__TRY
	_Ancestor.AddChildActivity(activity := _Ancestor);
__CATCH(exceptionCode)
	exception := TOF_Core.ExceptionManager.GetLastException(
		exceptionCode := exceptionCode,
		catchPointNamespaceName := NamespaceName,
		catchPointPOUName := __POUNAME(),
		catchPointPosition := __POSITION()
	);
	caught := __QUERYINTERFACE(exception, attachmentException);
__ENDTRY

assertions.ThatBool(actual := caught, message := "Self attachment must be rejected").IsTrue();
_Ancestor.AddChildActivity(activity := _Descendant);
caught := FALSE;

__TRY
	_Descendant.AddChildActivity(activity := _Ancestor);
__CATCH(exceptionCode)
	exception := TOF_Core.ExceptionManager.GetLastException(
		exceptionCode := exceptionCode,
		catchPointNamespaceName := NamespaceName,
		catchPointPOUName := __POUNAME(),
		catchPointPosition := __POSITION()
	);
	caught := __QUERYINTERFACE(exception, attachmentException);
__ENDTRY

assertions.ThatBool(actual := caught, message := "Ancestor attachment must be rejected").IsTrue();

_Pick.AddBranch(condition := _PickFirstCondition, activity := _PickFirstActivity);
caught := FALSE;

__TRY
	_Pick.AddBranch(condition := _PickFirstCondition, activity := _PickSecondActivity);
__CATCH(exceptionCode)
	exception := TOF_Core.ExceptionManager.GetLastException(
		exceptionCode := exceptionCode,
		catchPointNamespaceName := NamespaceName,
		catchPointPOUName := __POUNAME(),
		catchPointPosition := __POSITION()
	);
	caught := __QUERYINTERFACE(exception, attachmentException);
__ENDTRY

assertions.ThatBool(actual := caught, message := "A condition cannot occupy two branch slots").IsTrue();
caught := FALSE;

__TRY
	_Pick.AddBranch(condition := _PickSecondCondition, activity := _PickFirstActivity);
__CATCH(exceptionCode)
	exception := TOF_Core.ExceptionManager.GetLastException(
		exceptionCode := exceptionCode,
		catchPointNamespaceName := NamespaceName,
		catchPointPOUName := __POUNAME(),
		catchPointPosition := __POSITION()
	);
	caught := __QUERYINTERFACE(exception, attachmentException);
__ENDTRY

assertions.ThatBool(actual := caught, message := "An activity cannot occupy two branch slots").IsTrue();
actualElement := _PickSecondCondition.Parent;
assertions.ThatBool(
	actual := actualElement = 0,
	message := "Rejected pairs must not attach the unused condition"
).IsTrue();
actualElement := _PickSecondActivity.Parent;
assertions.ThatBool(
	actual := actualElement = 0,
	message := "Rejected pairs must not attach the unused activity"
).IsTrue();
_Pick.AddBranch(condition := _PickSecondCondition, activity := _PickSecondActivity);
_PickFirstActivity.completeRunning := TRUE;
_Pick.RequestStart();
assertions.ThatDInt(
	actual := _Pick.CurrentBranchIndex,
	message := "The original first pair must retain priority"
).ToBe(expected := 0);
assertions.ThatDInt(
	actual := _PickFirstActivity.startCount,
	message := "The first branch activity must start"
).ToBe(expected := 1);
assertions.ThatDInt(
	actual := _PickSecondActivity.startCount,
	message := "The second branch must remain unstarted"
).ToBe(expected := 0);

_SequenceFirst.completeRunning := TRUE;
_SequenceSecond.completeRunning := TRUE;
_Sequence.RequestStart();
_Sequence.Execute();
assertions.ThatBool(
	actual := _Sequence.State = TOF_Workflow.WORKFLOW_ELEMENT_STATE.PASSIVE_COMPLETED,
	message := "The original two valid slots must complete"
).IsTrue();
assertions.ThatDInt(
	actual := _SequenceFirst.startCount,
	message := "First child must start once"
).ToBe(expected := 1);
assertions.ThatDInt(
	actual := _SequenceSecond.startCount,
	message := "Second child must start once"
).ToBe(expected := 1);

_Sequence.RequestReset();
_Pick.RequestReset();
assertions.ThatBool(
	actual := _Sequence.CurrentActivityIndex = TOF_Workflow.Workflows.NO_SELECTED_ACTIVITY_INDEX,
	message := "Reset sequence must expose the documented absent-selection sentinel"
).IsTrue();
assertions.ThatBool(
	actual := _Pick.CurrentBranchIndex = TOF_Workflow.Workflows.NO_SELECTED_ACTIVITY_INDEX,
	message := "Reset branch selection must expose the same absent-selection sentinel"
).IsTrue();
END_METHOD

(*!
<summary>Preserves task internal-abort diagnostics while stopping.</summary>
<description>
Uses independently prepared persistent fixtures. Expected failures are checked by exception interface;
ordinary unexpected exceptions leave fixture ownership with the suite.
</description>
<param name="assertions">Valid assertion context borrowed from the active case.</param>
*)
METHOD PRIVATE testTaskAbortDuringSuspend
VAR_INPUT
	assertions : REFERENCE TO TOF_Testing.Assertions;
END_VAR
_SuspendAbortActivity.Configure(task := _SuspendAbortTask);
_SuspendAbortWorkflow.SetRootActivity(rootActivity := _SuspendAbortActivity);
_SuspendAbortWorkflow.RequestStart();
_SuspendAbortTask.processingResult := TOF_Tasks.TASK_PROCESSING_STATE.ABORTED;
_SuspendAbortWorkflow.RequestSuspend();
assertions.ThatBool(
	actual := _SuspendAbortActivity.State = TOF_Workflow.WORKFLOW_ELEMENT_STATE.PASSIVE_HALTED,
	message := "An internal abort while suspending must remain HALTED"
).IsTrue();
assertions.ThatWideString(
	actual := _SuspendAbortActivity.HaltReason,
	message := "The task abort reason must survive adapter translation"
).ToBe(expected := "Controlled task internal abort");
_SuspendAbortWorkflow.RequestReset();
END_METHOD

(*!
<summary>Preserves successful task completion when work finishes during suspension.</summary>
<description>
Uses independently prepared persistent fixtures. Expected failures are checked by exception interface;
ordinary unexpected exceptions leave fixture ownership with the suite.
</description>
<param name="assertions">Valid assertion context borrowed from the active case.</param>
*)
METHOD PRIVATE testTaskCompletionDuringSuspend
VAR_INPUT
	assertions : REFERENCE TO TOF_Testing.Assertions;
END_VAR
_SuspendDoneActivity.Configure(task := _SuspendDoneTask);
_SuspendDoneWorkflow.SetRootActivity(rootActivity := _SuspendDoneActivity);
_SuspendDoneWorkflow.RequestStart();
_SuspendDoneTask.processingResult := TOF_Tasks.TASK_PROCESSING_STATE.DONE;
_SuspendDoneWorkflow.RequestSuspend();
assertions.ThatBool(
	actual := _SuspendDoneActivity.State = TOF_Workflow.WORKFLOW_ELEMENT_STATE.PASSIVE_COMPLETED,
	message := "Work completed during suspension must retain its completion outcome"
).IsTrue();
_SuspendDoneWorkflow.RequestReset();
END_METHOD

(*!
<summary>Reports a task processing failure during suspension as an activity failure.</summary>
<description>
Uses independently prepared persistent fixtures. Expected failures are checked by exception interface;
ordinary unexpected exceptions leave fixture ownership with the suite.
</description>
<param name="assertions">Valid assertion context borrowed from the active case.</param>
*)
METHOD PRIVATE testTaskFailureDuringSuspend
VAR_INPUT
	assertions : REFERENCE TO TOF_Testing.Assertions;
END_VAR
_SuspendFailureActivity.Configure(task := _SuspendFailureTask);
_SuspendFailureWorkflow.SetRootActivity(rootActivity := _SuspendFailureActivity);
_SuspendFailureWorkflow.RequestStart();
_SuspendFailureTask.processingResult := TOF_Tasks.TASK_PROCESSING_STATE.ERROR;
_SuspendFailureWorkflow.RequestSuspend();

assertions.ThatBool(
	actual := _SuspendFailureTask.State.Stopped,
	message := "The failed task must reach STOPPED"
).IsTrue();
assertions.ThatBool(
	actual := _SuspendFailureActivity.State = TOF_Workflow.WORKFLOW_ELEMENT_STATE.PASSIVE_FAILED,
	message := "Task failure while suspending must not be reported as SUSPENDED"
).IsTrue();
assertions.ThatBool(
	actual := _SuspendFailureWorkflow.FailError.HasError,
	message := "Failure diagnostics must be retained"
).IsTrue();
_SuspendFailureWorkflow.RequestReset();
END_METHOD

(*!
<summary>
Keeps servicing cancellation through release and exposes a release failure with explicit resource recovery.
</summary>
<description>
Uses independently prepared persistent fixtures. Expected failures are checked by exception interface;
ordinary unexpected exceptions leave fixture ownership with the suite.
</description>
<param name="assertions">Valid assertion context borrowed from the active case.</param>
*)
METHOD PRIVATE testTaskReleaseFailureDuringCancel
VAR_INPUT
	assertions : REFERENCE TO TOF_Testing.Assertions;
END_VAR
VAR
	caught : BOOL;
	exceptionCode : __SYSTEM.ExceptionCode;
	exception : TOF_Core.IException;
	configurationException : TOF_Workflow.IWorkflowConfigurationException;
	i : INT;
END_VAR
_ReleaseTask.resource := _ReleaseResource;
_ReleaseActivity.Configure(task := _ReleaseTask);
_ReleaseWorkflow.SetRootActivity(rootActivity := _ReleaseActivity);
_ReleaseWorkflow.RequestStart();

FOR i := 1 TO 8 DO
	_ReleaseWorkflow.Execute();

	IF _ReleaseResource.ResourceAcquired THEN
		EXIT;
	END_IF
END_FOR

assertions.ThatBool(
	actual := _ReleaseResource.ResourceAcquired,
	message := "Synthetic acquisition must finish before cancellation"
).IsTrue();
_ReleaseResource.ThrowOnStartRelease := TRUE;
_ReleaseWorkflow.RequestCancel(reason := "Release failure test");
caught := FALSE;

__TRY
	_ReleaseActivity.Configure(task := _ReleaseReplacement);
__CATCH(exceptionCode)
	exception := TOF_Core.ExceptionManager.GetLastException(
		exceptionCode := exceptionCode,
		catchPointNamespaceName := NamespaceName,
		catchPointPOUName := __POUNAME(),
		catchPointPosition := __POSITION()
	);
	caught := __QUERYINTERFACE(exception, configurationException);
__ENDTRY

assertions.ThatBool(actual := caught, message := "Resource release must still block task replacement").IsTrue();
_ReleaseWorkflow.Execute();
assertions.ThatBool(
	actual := _ReleaseActivity.State = TOF_Workflow.WORKFLOW_ELEMENT_STATE.PASSIVE_FAILED,
	message := "Release failure must not become a successful cancellation"
).IsTrue();
assertions.ThatBool(
	actual := _ReleaseWorkflow.FailError.HasError,
	message := "Release failure diagnostics must remain visible"
).IsTrue();

// The synthetic manager intentionally retains ownership on failed release; recover it explicitly.
_ReleaseResource.ThrowOnStartRelease := FALSE;
_ReleaseResource.StartRelease();

FOR i := 1 TO 3 DO
	_ReleaseResource.Execute();
END_FOR

assertions.ThatBool(
	actual := _ReleaseResource.ResourceAcquired,
	message := "The test must release its synthetic resource"
).IsFalse();
_ReleaseWorkflow.RequestReset();
assertions.ThatBool(
	actual := _ReleaseActivity.State = TOF_Workflow.WORKFLOW_ELEMENT_STATE.PASSIVE_READY,
	message := "Explicit resource recovery must permit adapter reset"
).IsTrue();
END_METHOD

(*!
<summary>Resolves borrowed local and ancestor bindings and reports absence without changing storage.</summary>
<description>
Uses independently prepared persistent fixtures. Expected failures are checked by exception interface;
ordinary unexpected exceptions leave fixture ownership with the suite.
</description>
<param name="assertions">Valid assertion context borrowed from the active case.</param>
*)
METHOD PRIVATE testVariableLookup
VAR_INPUT
	assertions : REFERENCE TO TOF_Testing.Assertions;
END_VAR
VAR
	found : BOOL;
	resolved : TOF_Core.GENERIC_VALUE;
END_VAR
_LookupWorkflow.BindPlcVariable(name := 'Shared', plcVariable := _LookupWorkflowValue);
_LookupParent.BindPlcVariable(name := 'Shared', plcVariable := _LookupParentValue);
_LookupParent.AddChildActivity(activity := _LookupChild);
_LookupCondition.ParentActivity := _LookupChild;
_LookupCondition.BindPlcVariable(name := 'Local', plcVariable := _LookupConditionValue);

found := _LookupChild.TryGetVariable(name := 'Shared', variable => resolved);
assertions.ThatBool(actual := found, message := "A child must resolve its parent binding").IsTrue();
assertions.ThatBool(
	actual := resolved.Address = ADR(_LookupParentValue),
	message := "Parent binding precedes workflow fallback"
).IsTrue();
found := _LookupCondition.TryGetVariable(name := 'Shared', variable => resolved);
assertions.ThatBool(actual := found, message := "A condition must resolve its activity hierarchy").IsTrue();
assertions.ThatBool(
	actual := resolved.Address = ADR(_LookupParentValue),
	message := "Condition lookup must retain parent storage"
).IsTrue();
found := _LookupCondition.TryGetVariable(name := 'Local', variable => resolved);
assertions.ThatBool(actual := found, message := "A condition must resolve its own binding").IsTrue();
assertions.ThatBool(
	actual := resolved.Address = ADR(_LookupConditionValue),
	message := "Local lookup must retain condition storage"
).IsTrue();
found := _LookupCondition.TryGetVariable(name := 'Missing', variable => resolved);
assertions.ThatBool(actual := found, message := "Missing variables are a normal Try failure").IsFalse();
END_METHOD

(*!
<summary>Rejects foreign activities and conditions through every construction family.</summary>
<description>
Uses independently prepared persistent fixtures. Expected failures are checked by exception interface;
ordinary unexpected exceptions leave fixture ownership with the suite.
</description>
<param name="assertions">Valid assertion context borrowed from the active case.</param>
*)
METHOD PRIVATE testWorkflowIsolation
VAR_INPUT
	assertions : REFERENCE TO TOF_Testing.Assertions;
END_VAR
VAR
	expectedWorkflow : TOF_Workflow.IWorkflow;
	actualElement : TOF_Workflow.IWorkflowElement;
	actualWorkflow : TOF_Workflow.IWorkflow;
	caught : BOOL;
	exceptionCode : __SYSTEM.ExceptionCode;
	exception : TOF_Core.IException;
	attachmentException : TOF_Workflow.IWorkflowAttachmentException;
END_VAR
caught := FALSE;

__TRY
	_IsolationSequence.AddChildActivity(activity := _ForeignChild);
__CATCH(exceptionCode)
	exception := TOF_Core.ExceptionManager.GetLastException(
		exceptionCode := exceptionCode,
		catchPointNamespaceName := NamespaceName,
		catchPointPOUName := __POUNAME(),
		catchPointPosition := __POSITION()
	);
	caught := __QUERYINTERFACE(exception, attachmentException);
__ENDTRY

assertions.ThatBool(actual := caught, message := "Sequence must reject a foreign child").IsTrue();
caught := FALSE;

__TRY
	_IsolationParallel.AddChildActivity(activity := _ForeignChild);
__CATCH(exceptionCode)
	exception := TOF_Core.ExceptionManager.GetLastException(
		exceptionCode := exceptionCode,
		catchPointNamespaceName := NamespaceName,
		catchPointPOUName := __POUNAME(),
		catchPointPosition := __POSITION()
	);
	caught := __QUERYINTERFACE(exception, attachmentException);
__ENDTRY

assertions.ThatBool(actual := caught, message := "Parallel must reject a foreign child").IsTrue();
caught := FALSE;

__TRY
	_IsolationWait.Configure(condition := _ForeignCondition);
__CATCH(exceptionCode)
	exception := TOF_Core.ExceptionManager.GetLastException(
		exceptionCode := exceptionCode,
		catchPointNamespaceName := NamespaceName,
		catchPointPOUName := __POUNAME(),
		catchPointPosition := __POSITION()
	);
	caught := __QUERYINTERFACE(exception, attachmentException);
__ENDTRY

assertions.ThatBool(actual := caught, message := "WaitCondition must reject a foreign condition").IsTrue();
caught := FALSE;

__TRY
	_IsolationWhile.Configure(condition := _ForeignCondition, body := 0);
__CATCH(exceptionCode)
	exception := TOF_Core.ExceptionManager.GetLastException(
		exceptionCode := exceptionCode,
		catchPointNamespaceName := NamespaceName,
		catchPointPOUName := __POUNAME(),
		catchPointPosition := __POSITION()
	);
	caught := __QUERYINTERFACE(exception, attachmentException);
__ENDTRY

assertions.ThatBool(actual := caught, message := "While must reject a foreign condition").IsTrue();
caught := FALSE;

__TRY
	_IsolationIf.Configure(condition := _ForeignCondition, trueActivity := 0, falseActivity := 0);
__CATCH(exceptionCode)
	exception := TOF_Core.ExceptionManager.GetLastException(
		exceptionCode := exceptionCode,
		catchPointNamespaceName := NamespaceName,
		catchPointPOUName := __POUNAME(),
		catchPointPosition := __POSITION()
	);
	caught := __QUERYINTERFACE(exception, attachmentException);
__ENDTRY

assertions.ThatBool(actual := caught, message := "IfElse must reject a foreign condition").IsTrue();
caught := FALSE;

__TRY
	_IsolationNot.Configure(condition := _ForeignCondition);
__CATCH(exceptionCode)
	exception := TOF_Core.ExceptionManager.GetLastException(
		exceptionCode := exceptionCode,
		catchPointNamespaceName := NamespaceName,
		catchPointPOUName := __POUNAME(),
		catchPointPosition := __POSITION()
	);
	caught := __QUERYINTERFACE(exception, attachmentException);
__ENDTRY

assertions.ThatBool(actual := caught, message := "Not must reject a foreign condition").IsTrue();
caught := FALSE;

__TRY
	_IsolationGroup.AddChildCondition(condition := _ForeignCondition);
__CATCH(exceptionCode)
	exception := TOF_Core.ExceptionManager.GetLastException(
		exceptionCode := exceptionCode,
		catchPointNamespaceName := NamespaceName,
		catchPointPOUName := __POUNAME(),
		catchPointPosition := __POSITION()
	);
	caught := __QUERYINTERFACE(exception, attachmentException);
__ENDTRY

assertions.ThatBool(actual := caught, message := "CompositeCondition must reject a foreign condition").IsTrue();
caught := FALSE;

__TRY
	_UnassociatedSequence.AddChildActivity(activity := _ForeignChild);
__CATCH(exceptionCode)
	exception := TOF_Core.ExceptionManager.GetLastException(
		exceptionCode := exceptionCode,
		catchPointNamespaceName := NamespaceName,
		catchPointPOUName := __POUNAME(),
		catchPointPosition := __POSITION()
	);
	caught := __QUERYINTERFACE(exception, attachmentException);
__ENDTRY

assertions.ThatBool(
	actual := caught,
	message := "An unassociated subtree cannot hide an explicitly owned child"
).IsTrue();
actualElement := _ForeignChild.Parent;
assertions.ThatBool(actual := actualElement = 0, message := "Foreign activity must remain unattached").IsTrue();
actualElement := _ForeignCondition.Parent;
assertions.ThatBool(actual := actualElement = 0, message := "Foreign condition must remain unattached").IsTrue();

expectedWorkflow := _IsolationWorkflow;
_UnassociatedSequence.AddChildActivity(activity := _UnassociatedChild);
_IsolationSequence.AddChildActivity(activity := _UnassociatedSequence);
actualWorkflow := _UnassociatedChild.Workflow;
assertions.ThatBool(
	actual := actualWorkflow = expectedWorkflow,
	message := "An entirely unassociated subtree must inherit its attached parent owner"
).IsTrue();
END_METHOD

(*!
<summary>Checks owned values through two loop iterations, a nested condition and a workflow reset.</summary>
<description>Advances the loop through body completion and the next iteration before checking restored values.</description>
<param name="assertions">Valid assertion context borrowed from the active case.</param>
*)
METHOD PRIVATE testDeclaredVariableReset
VAR_INPUT
	assertions : REFERENCE TO TOF_Testing.Assertions;
END_VAR
VAR
	initial : UINT := 7;
	changed : UINT := 23;
	initialText : WSTRING(24) := "Start";
	workflowCount : TOF_Core.GENERIC_VALUE;
	loopCount : TOF_Core.GENERIC_VALUE;
	bodyCount : TOF_Core.GENERIC_VALUE;
	textValue : TOF_Core.GENERIC_VALUE;
	found : BOOL;
	i : DINT;
END_VAR
_DeclarationLoop.Configure(condition := _DeclarationGuard, body := _DeclarationBody);
_DeclarationBody.completeRunning := TRUE;
_DeclarationGroup.Configure(condition := _DeclarationLeaf);
_DeclarationGroup.ParentActivity := _DeclarationBody;

_DeclarationWorkflow.DeclareVariable(name := 'Count', initialValue := initial);
_DeclarationLoop.DeclareVariable(name := 'Count', initialValue := initial);
_DeclarationBody.DeclareVariable(name := 'Count', initialValue := initial);
_DeclarationLeaf.DeclareVariable(name := 'Text', initialValue := initialText);
_DeclarationBody.BindPlcVariable(name := 'Input', plcVariable := _DeclarationInput);
_DeclarationWorkflow.SetRootActivity(rootActivity := _DeclarationLoop);
initial := 99;
initialText := "Changed";

found := _DeclarationWorkflow.TryGetVariable(name := 'Count', variable => workflowCount)
	AND_THEN _DeclarationLoop.TryGetLocalVariable(name := 'Count', variable => loopCount)
	AND_THEN _DeclarationGroup.TryGetVariable(name := 'Count', variable => bodyCount)
	AND_THEN _DeclarationLeaf.TryGetLocalVariable(name := 'Text', variable => textValue);
assertions.ThatBool(
	actual := found,
	message := "All declarations must resolve from their configured scopes"
).IsTrue();

IF found THEN
	assertions.ThatBool(
		actual := workflowCount.Address <> loopCount.Address AND_THEN loopCount.Address <> bodyCount.Address
			AND_THEN bodyCount.Address <> workflowCount.Address AND_THEN bodyCount.Address <> ADR(initial),
		message := "Equal names in separate scopes must keep independent storage"
	).IsTrue();
	assertions.ThatBool(
		actual := NOT workflowCount.IsMemoryOwner AND_THEN NOT loopCount.IsMemoryOwner
			AND_THEN NOT bodyCount.IsMemoryOwner AND_THEN NOT textValue.IsMemoryOwner,
		message := "Resolved declarations must be borrowed"
	).IsTrue();
	assertions.ThatBool(
		actual := textValue.Size = XSIZEOF(initialText) AND_THEN textValue.AsWStringReference() = "Start",
		message := "Owned strings must preserve initial contents and full declared capacity"
	).IsTrue();

	_DeclarationWorkflow.RequestStart();
	workflowCount.ChangeValueByAny(value := changed);
	loopCount.ChangeValueByAny(value := changed);
	bodyCount.ChangeValueByAny(value := changed);
	textValue.ChangeValueByAny(value := initialText);
	_DeclarationInput := changed;

	_DeclarationWorkflow.Execute();
	_DeclarationWorkflow.Execute();
	assertions.ThatBool(
		actual := _DeclarationBody.startCount = 2,
		message := "The loop must restart its body"
	).IsTrue();
	assertions.ThatBool(
		actual := bodyCount.AsUInt() = 7 AND_THEN textValue.AsWStringReference() = "Start",
		message := "Body and nested condition must restore in place between iterations"
	).IsTrue();
	assertions.ThatBool(
		actual := loopCount.AsUInt() = changed AND_THEN workflowCount.AsUInt() = changed,
		message := "Resetting the body must preserve the loop and workflow variables"
	).IsTrue();

	_DeclarationWorkflow.RequestCancel(reason := "End declaration test");

	FOR i := 1 TO 4 DO
		IF _DeclarationWorkflow.Busy THEN
			_DeclarationWorkflow.Execute();
		END_IF
	END_FOR

	_DeclarationBody.deferFirstResetStep := TRUE;
	bodyCount.ChangeValueByAny(value := changed);
	_DeclarationWorkflow.RequestReset();

	assertions.ThatBool(
		actual := _DeclarationWorkflow.State = TOF_Workflow.WORKFLOW_ELEMENT_STATE.ACTIVE_RESETTING
			AND_THEN workflowCount.AsUInt() = changed AND_THEN bodyCount.AsUInt() = changed,
		message := "A pending reset must preserve current values until its owner completes"
	).IsTrue();

	FOR i := 1 TO 4 DO
		IF _DeclarationWorkflow.Busy THEN
			_DeclarationWorkflow.Execute();
		END_IF
	END_FOR

	assertions.ThatBool(
		actual := _DeclarationWorkflow.State = TOF_Workflow.WORKFLOW_ELEMENT_STATE.PASSIVE_READY
			AND_THEN workflowCount.AsUInt() = 7 AND_THEN loopCount.AsUInt() = 7 AND_THEN bodyCount.AsUInt() = 7,
		message := "Successful workflow reset must restore workflow and loop declarations"
	).IsTrue();
	assertions.ThatBool(
		actual := _DeclarationInput = changed,
		message := "Reset must preserve borrowed PLC storage"
	).IsTrue();
END_IF
END_METHOD

(*!
<summary>Checks duplicate, empty and composite declarations without replacing existing local storage.</summary>
<param name="assertions">Valid assertion context borrowed from the active case.</param>
*)
METHOD PRIVATE testDeclaredVariableValidation
VAR_INPUT
	assertions : REFERENCE TO TOF_Testing.Assertions;
END_VAR
VAR
	initial : UINT := 4;
	recordValue : TOF_Core.GENERIC_KEY_VALUE_PAIR;
	workflow : TOF_Workflow.IWorkflow;
	declarations : TOF_Workflow.IDeclaredVariableContainer;
	resolved : TOF_Core.GENERIC_VALUE;
	found : BOOL;
	caught : BOOL;
	exceptionCode : __SYSTEM.ExceptionCode;
	exception : TOF_Core.IException;
	configurationError : TOF_Workflow.IWorkflowConfigurationException;
	i : DINT;
END_VAR
workflow := _DeclarationValidation;
found := __QUERYINTERFACE(workflow, declarations);
assertions.ThatBool(actual := found, message := "Standard workflow must expose the declaration capability").IsTrue();

IF NOT found THEN
	RETURN;
END_IF

_DeclarationValidation.BindPlcVariable(name := 'Borrowed', plcVariable := _DeclarationInput);
declarations.DeclareVariable(name := 'Owned', initialValue := initial);

FOR i := 1 TO 5 DO
	caught := FALSE;

	__TRY
		CASE i OF
			1:
				_DeclarationValidation.DeclareVariable(name := 'Borrowed', initialValue := initial);
			2:
				_DeclarationValidation.BindPlcVariable(name := 'Owned', plcVariable := _DeclarationInput);
			3:
				_DeclarationValidation.DeclareVariable(name := 'Owned', initialValue := initial);
			4:
				_DeclarationValidation.DeclareVariable(name := '', initialValue := initial);
			5:
				_DeclarationValidation.DeclareVariable(name := 'Invalid', initialValue := recordValue);
		END_CASE
	__CATCH(exceptionCode)
		exception := TOF_Core.ExceptionManager.GetLastException(
			exceptionCode := exceptionCode,
			catchPointNamespaceName := NamespaceName,
			catchPointPOUName := __POUNAME(),
			catchPointPosition := __POSITION()
		);
		caught := __QUERYINTERFACE(exception, configurationError);
	__ENDTRY

	assertions.ThatBool(
		actual := caught,
		message := "Each invalid declaration must raise a configuration error"
	).IsTrue();
END_FOR

found := _DeclarationValidation.TryGetVariable(name := 'Owned', variable => resolved);
assertions.ThatBool(
	actual := found AND_THEN resolved.AsUInt() = initial,
	message := "Rejected replacement preserves value"
).IsTrue();
found := _DeclarationValidation.TryGetVariable(name := 'Borrowed', variable => resolved);
assertions.ThatBool(
	actual := found AND_THEN resolved.Address = ADR(_DeclarationInput),
	message := "Borrowed binding survives"
).IsTrue();
found := _DeclarationValidation.TryGetVariable(name := 'Invalid', variable => resolved);
assertions.ThatBool(actual := found, message := "Rejected type must leave the scope unchanged").IsFalse();
END_METHOD

(*!
<summary>Checks the diagnostic target order and the transition predicate for every lifecycle state pair.</summary>
<description>Uses independent expected lists and passes each candidate as the compatibility argument.</description>
<param name="assertions">Valid assertion context borrowed from the active case.</param>
*)
METHOD PRIVATE testTransitionDiagnostics
VAR_INPUT
	assertions : REFERENCE TO TOF_Testing.Assertions;
END_VAR
VAR CONSTANT
	states : ARRAY [0..9] OF TOF_Workflow.WORKFLOW_ELEMENT_STATE := [
		TOF_Workflow.WORKFLOW_ELEMENT_STATE.PASSIVE_READY,
		TOF_Workflow.WORKFLOW_ELEMENT_STATE.PASSIVE_COMPLETED,
		TOF_Workflow.WORKFLOW_ELEMENT_STATE.PASSIVE_HALTED,
		TOF_Workflow.WORKFLOW_ELEMENT_STATE.PASSIVE_CANCELLED,
		TOF_Workflow.WORKFLOW_ELEMENT_STATE.PASSIVE_FAILED,
		TOF_Workflow.WORKFLOW_ELEMENT_STATE.PASSIVE_SUSPENDED,
		TOF_Workflow.WORKFLOW_ELEMENT_STATE.ACTIVE_RUNNING,
		TOF_Workflow.WORKFLOW_ELEMENT_STATE.ACTIVE_CANCELLING,
		TOF_Workflow.WORKFLOW_ELEMENT_STATE.ACTIVE_SUSPENDING,
		TOF_Workflow.WORKFLOW_ELEMENT_STATE.ACTIVE_RESETTING
	];
	expectedNames : ARRAY [0..9] OF STRING(255) := [
		'ACTIVE_RUNNING',
		'ACTIVE_RESETTING',
		'ACTIVE_RESETTING',
		'ACTIVE_RESETTING',
		'ACTIVE_RESETTING',
		'ACTIVE_RUNNING,ACTIVE_CANCELLING',
		'PASSIVE_COMPLETED,ACTIVE_SUSPENDING,ACTIVE_CANCELLING,PASSIVE_HALTED,PASSIVE_FAILED',
		'PASSIVE_CANCELLED,PASSIVE_COMPLETED,PASSIVE_HALTED,PASSIVE_FAILED',
		'PASSIVE_SUSPENDED,PASSIVE_COMPLETED,PASSIVE_HALTED,PASSIVE_FAILED',
		'PASSIVE_READY,PASSIVE_FAILED'
	];
END_VAR
VAR
	i : DINT;
	j : DINT;
	actualNames : STRING(255);
	expectedList : STRING(255);
	targetToken : STRING;
	permitted : BOOL;
END_VAR
FOR i := LOWER_BOUND(states, 1) TO UPPER_BOUND(states, 1) DO
	expectedList := TOF_Core.Strings.Concat255(',', expectedNames[i], ',');

	FOR j := LOWER_BOUND(states, 1) TO UPPER_BOUND(states, 1) DO
		actualNames := TOF_Workflow.Workflows.GetAllowedTransitionNames(currentState := states[i]);
		assertions.ThatBool(
			actual := actualNames = expectedNames[i],
			message := TO_WSTRING(TOF_Core.Strings.Concat255('Diagnostic order for ', TO_STRING(states[i])))
		).IsTrue();
		targetToken := TOF_Core.Strings.Concat255(',', TO_STRING(states[j]), ',');
		permitted := TOF_Workflow.Workflows.ValidateTransition(currentState := states[i], newState := states[j]);
		// SA0175: Exact ASCII token search within the comma-delimited diagnostic transition list.
		{analysis -175}
		assertions.ThatBool(
			actual := permitted = (Tc2_Standard.FIND(STR1 := expectedList, STR2 := targetToken) > 0),
			message := TO_WSTRING(TOF_Core.Strings.Concat255('Transition from ', TO_STRING(states[i]), ' to ', TO_STRING(states[j])))
		).IsTrue();
		{analysis +175}
	END_FOR
END_FOR
END_METHOD

(*!
<summary>Provides the application-specific test activity to the workflow factory.</summary>
<description>Returns zero for unknown names. The suite owns the disposal counter until the registered child exits.</description>
<param name="typeName">Requested type.</param>
<param name="workflow">Prospective owner.</param>
*)
METHOD CreateElement : TOF_Workflow.IWorkflowElement
VAR_INPUT
	typeName : STRING(255);
	workflow : TOF_Workflow.IWorkflow;
END_VAR
VAR
	created : POINTER TO WorkflowContractActivity;
END_VAR
IF typeName <> TOF_Core.Strings.Concat255(CurrentNamespace.Name, '.WorkflowContractActivity') THEN
	RETURN;
END_IF

created := __NEW(WorkflowContractActivity(workflow := workflow));

IF created = 0 THEN
	TOF_Core.DynamicMemoryManager.RaiseAllocationFailure();
END_IF

created^.exitCount REF= _FactoryExits;
created^.completeRunning := TRUE;
CreateElement := created^;
END_METHOD

(*!
<summary>Builds a mixed factory tree and observes array declaration, mutation, reset and disposal.</summary>
<description>Uses persistent workflow ownership and synthetic values in one task.</description>
<param name="assertions">Valid assertion context borrowed from the active case.</param>
*)
METHOD PRIVATE testFactoryDeclarations
VAR_INPUT
	assertions : REFERENCE TO TOF_Testing.Assertions;
END_VAR
VAR
	element : TOF_Workflow.IWorkflowElement;
	sequence : TOF_Workflow.ISequenceActivity;
	child : TOF_Workflow.IActivity;
	scope : TOF_Workflow.IDeclaredVariableContainer;
	binder : TOF_Workflow.IVariableBinder;
	initials : ARRAY [3..4] OF __SYSTEM.AnyType;
	firstValue : BYTE := BYTE#2;
	secondValue : BYTE := BYTE#5;
	initialCopy : BYTE;
	position : DINT;
	declarationCount : DINT;
	bindingName : STRING;
	declaration : TOF_Workflow.VARIABLE_DECLARATION;
	live : TOF_Core.GENERIC_VALUE;
	found : BOOL;
	ready : BOOL;
END_VAR
__TRY
	element := TOF_Workflow.Workflows.CreateElement(
		typeName := 'TOF_Workflow.SequenceActivity',
		workflow := _FactoryWorkflow
	);
	ready := __QUERYINTERFACE(element, sequence);
	element := TOF_Workflow.Workflows.CreateElement(
		typeName := TOF_Core.Strings.Concat255(CurrentNamespace.Name, '.WorkflowContractActivity'),
		workflow := _FactoryWorkflow,
		factory := THIS^
	);
	ready := ready
		AND_THEN __QUERYINTERFACE(element, child)
		AND_THEN __QUERYINTERFACE(element, scope)
		AND_THEN __QUERYINTERFACE(element, binder);
	assertions.ThatBool(
		actual := ready,
		message := "Built-in and custom factories must return the requested node capabilities"
	).IsTrue();

	IF ready THEN
		sequence.AddChildActivity(activity := child);
		_FactoryWorkflow.SetRootActivity(rootActivity := sequence);
		binder.BindPlcVariable(name := 'Input', plcVariable := _DeclarationInput);
		initials[3] := TOF_Workflow.Workflows.GetValueDescriptor(value := firstValue);
		initials[4] := TOF_Workflow.Workflows.GetValueDescriptor(value := secondValue);
		scope.DeclareArray(name := 'Limits', initialValues := ADR(initials[3]), elementCount := 2);
		scope.DeclareVariable(name := 'Flags', initialValue := firstValue);
		firstValue := BYTE#255;
		found := FALSE;

		WHILE scope.NextDeclaration(position := position, name => bindingName, declaration => declaration) DO
			declarationCount := declarationCount + 1;
			assertions.ThatBool(
				actual := declaration.ElementType = __SYSTEM.TYPE_CLASS.TYPE_BYTE AND_THEN declaration.ElementSize = 1,
				message := "BYTE must preserve its exact IEC type"
			).IsTrue();

			IF bindingName = 'Limits' THEN
				found := declaration.IsArray AND_THEN declaration.ElementCount = 2;
			ELSE
				assertions.ThatBool(
					actual := bindingName = 'Flags' AND_THEN NOT declaration.IsArray AND_THEN declaration.ElementCount = 1,
					message := "Only local declarations must be enumerated"
				).IsTrue();
			END_IF
		END_WHILE

		assertions.ThatBool(
			actual := found AND_THEN declarationCount = 2,
			message := "Enumeration must include the array and scalar"
		).IsTrue();
		live := scope.GetDeclaredElement(name := 'Limits', index := 1);
		live.ChangeValueByAny(value := firstValue);
		scope.CopyInitialElement(
			name := 'Limits',
			index := 1,
			destination := TOF_Workflow.Workflows.GetValueDescriptor(value := initialCopy)
		);
		assertions.ThatBool(
			actual := initialCopy = BYTE#5 AND_THEN live.AsByte() = BYTE#255 AND_THEN NOT live.IsMemoryOwner,
			message := "Initial value and writable current element must be independent"
		).IsTrue();
		_FactoryWorkflow.RequestStart();
		_FactoryWorkflow.RequestReset();
		assertions.ThatBool(
			actual := live.AsByte() = BYTE#5,
			message := "Workflow reset must restore an owned array in place"
		).IsTrue();
		live := scope.GetDeclaredElement(name := 'Limits', index := 0);
		assertions.ThatBool(
			actual := live.AsByte() = BYTE#2,
			message := "Source bounds must map to zero-based declaration indices"
		).IsTrue();
	END_IF
__CATCH
	assertions.ThatBool(
		actual := FALSE,
		message := "Unexpected exception while building or exercising factory graph"
	).IsTrue();
__ENDTRY

_FactoryWorkflow.DisposeDynamicChildren();
TOF_Core.DynamicMemoryManager.RaiseIfAllocationFailed();
assertions.ThatBool(
	actual := _FactoryExits = 1,
	message := "Workflow disposal must invoke the custom child destructor once"
).IsTrue();
END_METHOD

(*!
<summary>Checks singleton shape and rejects invalid declarations, indices, destinations and unknown factory types.</summary>
<description>Uses persistent workflow ownership and synthetic values in one task.</description>
<param name="assertions">Valid assertion context borrowed from the active case.</param>
*)
METHOD PRIVATE testArrayValidation
VAR_INPUT
	assertions : REFERENCE TO TOF_Testing.Assertions;
END_VAR
VAR
	single : ARRAY [0..0] OF __SYSTEM.AnyType;
	mixed : ARRAY [0..1] OF __SYSTEM.AnyType;
	flag : BYTE := BYTE#1;
	number : USINT := USINT#42;
	element : TOF_Core.GENERIC_VALUE;
	node : TOF_Workflow.IWorkflowElement;
	position : DINT;
	bindingName : STRING;
	declaration : TOF_Workflow.VARIABLE_DECLARATION;
	more : BOOL;
	caught : BOOL;
	exceptionCode : __SYSTEM.ExceptionCode;
	exception : TOF_Core.IException;
	configurationError : TOF_Workflow.IWorkflowConfigurationException;
	i : DINT;
END_VAR
single[0] := TOF_Workflow.Workflows.GetValueDescriptor(value := flag);
_ArrayValidation.DeclareArray(name := 'One', initialValues := ADR(single[0]), elementCount := 1);
more := _ArrayValidation.NextDeclaration(position := position, name => bindingName, declaration => declaration);
assertions.ThatBool(
	actual := more AND_THEN declaration.IsArray AND_THEN declaration.ElementCount = 1,
	message := "A one-element array must preserve its shape"
).IsTrue();
mixed[0] := single[0];
mixed[1] := TOF_Workflow.Workflows.GetValueDescriptor(value := number);

FOR i := 1 TO 7 DO
	caught := FALSE;

	__TRY
		CASE i OF
			1:
				_ArrayValidation.DeclareArray(name := 'Bad', initialValues := ADR(mixed[0]), elementCount := 2);
			2:
				_ArrayValidation.DeclareArray(name := 'Bad', initialValues := 0, elementCount := 0);
			3:
				element := _ArrayValidation.GetDeclaredElement(name := 'One', index := -1);
			4:
				element := _ArrayValidation.GetDeclaredElement(name := 'One', index := 1);
			5:
				_ArrayValidation.CopyInitialElement(
					name := 'One',
					index := 0,
					destination := TOF_Workflow.Workflows.GetValueDescriptor(value := number)
				);
			6:
				node := TOF_Workflow.Workflows.CreateElement(
					typeName := 'Missing.Type',
					workflow := _ArrayValidation,
					factory := THIS^
				);
			7:
				_ArrayValidation.DeclareVariable(name := 'One', initialValue := number);
		END_CASE
	__CATCH(exceptionCode)
		exception := TOF_Core.ExceptionManager.GetLastException(
			exceptionCode := exceptionCode,
			catchPointNamespaceName := NamespaceName,
			catchPointPOUName := __POUNAME(),
			catchPointPosition := __POSITION()
		);
		caught := __QUERYINTERFACE(exception, configurationError);
	__ENDTRY

	assertions.ThatBool(
		actual := caught,
		message := "Invalid declaration, element access or factory name must raise"
	).IsTrue();
END_FOR

more := _ArrayValidation.NextDeclaration(position := position, name => bindingName, declaration => declaration);
assertions.ThatBool(actual := more, message := "Invalid definitions must not add dictionary entries").IsFalse();
assertions.ThatBool(
	actual := number = USINT#42,
	message := "Incorrect destination type must leave its bytes unchanged"
).IsTrue();
_ArrayValidation.DisposeDynamicChildren();
END_METHOD

(*!
<summary>Checks nested workflow serialization and the shape of a singleton array.</summary>
<description>Parses the actual output and checks the original value after modifying the live declaration.</description>
<param name="assertions">Valid assertion context borrowed from the active case.</param>
*)
METHOD PRIVATE testWriteConfiguration
VAR_INPUT
	assertions : REFERENCE TO TOF_Testing.Assertions;
END_VAR
VAR
	initial : UINT := 5;
	element : __SYSTEM.AnyType;
	live : TOF_Core.GENERIC_VALUE;
	number : POINTER TO UINT;
	document : Tc3_JsonXml.SJsonValue;
	field : Tc3_JsonXml.SJsonValue;
END_VAR
_WriteSequence.AddChildActivity(activity := _WriteDelay);
_WriteWorkflow.SetRootActivity(rootActivity := _WriteSequence);
element := TOF_Workflow.Workflows.GetValueDescriptor(value := initial);
_WriteDelay.DeclareArray(name := 'Limits', initialValues := ADR(element), elementCount := 1);
live := _WriteDelay.GetDeclaredElement(name := 'Limits', index := 0);
number := live.Address;
number^ := 9;
_ConfigWriter.Serialize(source := _WriteWorkflow, document := _ConfigDocument);
document := _ConfigParser.ParseDocument(sJson := _ConfigDocument);
field := _ConfigParser.FindMember(v := document, member := 'root');
field := _ConfigParser.FindMember(v := field, member := 'children');
assertions.ThatBool(
	actual := _ConfigParser.IsArray(v := field),
	message := "Sequence children must be an array"
).IsTrue();
field := _ConfigParser.GetArrayValueByIdx(v := field, idx := 0);
field := _ConfigParser.FindMember(v := field, member := 'variables');
field := _ConfigParser.GetArrayValueByIdx(v := field, idx := 0);
field := _ConfigParser.FindMember(v := field, member := 'initialValue');
assertions.ThatBool(
	actual := _ConfigParser.GetArraySize(v := field) = 1,
	message := "Preserve singleton array shape"
).IsTrue();
field := _ConfigParser.GetArrayValueByIdx(v := field, idx := 0);
assertions.ThatBool(
	actual := _ConfigParser.GetUint(v := field) = 5,
	message := "Serialize the reset image"
).IsTrue();
END_METHOD

(*!
<summary>Checks exclusive embedded ownership and shared external serialization.</summary>
<description>Uses a dual-interface object to verify that duplicate detection uses object identity.</description>
<param name="assertions">Valid assertion context borrowed from the active case.</param>
*)
METHOD PRIVATE testDependencyBindings
VAR_INPUT
	assertions : REFERENCE TO TOF_Testing.Assertions;
END_VAR
VAR
	instance : POINTER TO WorkflowBindingTask;
	otherInstance : POINTER TO WorkflowBindingTask;
	expectedComparer : TOF_Core.IComparer;
	actualComparer : TOF_Core.IComparer;
	exceptionCode : __SYSTEM.ExceptionCode;
	exception : TOF_Core.IException;
	configurationError : TOF_Workflow.IWorkflowConfigurationException;
	rejected : BOOL;
	document : Tc3_JsonXml.SJsonValue;
	binding : Tc3_JsonXml.SJsonValue;
	keyField : Tc3_JsonXml.SJsonValue;
END_VAR
_BindingFirst.ConfigureExternalTask(task := _BindingExternal, key := 'axis');
_BindingSecond.ConfigureExternalTask(task := _BindingExternal, key := 'axis');
_BindingComparer.ConfigureExternalComparer(comparer := _BindingExternal, key := 'axis');
_ConfigWriter.Serialize(source := _BindingSecond, document := _ConfigDocument);
document := _ConfigParser.ParseDocument(sJson := _ConfigDocument);
binding := _ConfigParser.FindMember(v := document, member := 'task');
keyField := _ConfigParser.FindMember(v := binding, member := 'key');
assertions.ThatBool(
	actual := _ConfigParser.GetString(v := keyField) = 'axis',
	message := "Keep the external key"
).IsTrue();
assertions.ThatBool(
	actual := _ConfigParser.FindMember(v := binding, member := 'type') = 0,
	message := "External task is borrowed"
).IsTrue();

instance := __NEW(WorkflowBindingTask(name := "Embedded"));

IF instance = 0 THEN
	TOF_Core.DynamicMemoryManager.RaiseAllocationFailure();
END_IF

_BindingFirst.ConfigureEmbeddedTask(task := instance^);

__TRY
	_BindingComparer.ConfigureEmbeddedComparer(comparer := instance^);
__CATCH(exceptionCode)
	exception := TOF_Core.ExceptionManager.GetLastException(
		exceptionCode := exceptionCode,
		catchPointNamespaceName := NamespaceName,
		catchPointPOUName := __POUNAME(),
		catchPointPosition := __POSITION()
	);
	rejected := __QUERYINTERFACE(exception, configurationError);
__ENDTRY

expectedComparer := _BindingExternal;
assertions.ThatBool(actual := rejected, message := "Reject second slot even through another interface").IsTrue();
actualComparer := _BindingComparer.Comparer;
assertions.ThatBool(
	actual := actualComparer = expectedComparer,
	message := "Keep previous external comparer"
).IsTrue();

otherInstance := __NEW(WorkflowBindingTask(name := "Another instance"));

IF otherInstance = 0 THEN
	TOF_Core.DynamicMemoryManager.RaiseAllocationFailure();
END_IF

_BindingComparer.ConfigureEmbeddedComparer(comparer := otherInstance^);
expectedComparer := otherInstance^;
actualComparer := _BindingComparer.Comparer;
assertions.ThatBool(
	actual := actualComparer = expectedComparer,
	message := "Allow another instance of the same type"
).IsTrue();

_ConfigWriter.Serialize(source := _BindingFirst, document := _ConfigDocument);
document := _ConfigParser.ParseDocument(sJson := _ConfigDocument);
binding := _ConfigParser.FindMember(v := document, member := 'task');
assertions.ThatBool(
	actual := _ConfigParser.FindMember(v := binding, member := 'configuration') <> 0,
	message := "Embed configuration"
).IsTrue();
assertions.ThatBool(
	actual := _ConfigParser.FindMember(v := binding, member := 'key') = 0,
	message := "Embedded task has no key"
).IsTrue();
_BindingWorkflow.DisposeDynamicChildren();
END_METHOD

(*!
<summary>Creates a fresh unowned dynamic embedded dependency for configuration loading.</summary>
<description>Returns zero for unknown type names.</description>
<param name="typeName">Requested qualified type name.</param>
*)
METHOD CreateDependency : TOF_Core.IObject
VAR_INPUT
	typeName : STRING(255);
END_VAR
VAR
	created : POINTER TO WorkflowBindingTask;
END_VAR
IF typeName <> TOF_Core.Strings.Concat255(CurrentNamespace.Name, '.WorkflowBindingTask') THEN
	RETURN;
END_IF

created := __NEW(WorkflowBindingTask(name := ""));

IF created = 0 THEN
	TOF_Core.DynamicMemoryManager.RaiseAllocationFailure();
END_IF

CreateDependency := created^;
END_METHOD

(*!
<summary>Resolves the shared external test dependency by its stable key.</summary>
<description>Returns zero for unknown keys.</description>
<param name="key">Requested external dependency key.</param>
*)
METHOD ResolveExternal : TOF_Core.IObject
VAR_INPUT
	key : STRING;
END_VAR
IF key = 'axis' THEN
	ResolveExternal := _BindingExternal;
END_IF
END_METHOD

(*!
<summary>Registers the external PLC variable on the freshly loaded workflow when enabled.</summary>
<description>Used to test both unresolved-variable rollback and successful binding.</description>
<param name="workflow">Fresh workflow being loaded.</param>
*)
METHOD BindVariables
VAR_INPUT
	workflow : TOF_Workflow.IWorkflow;
END_VAR
IF _BindLoadVariables THEN
	workflow.BindPlcVariable(name := 'External', plcVariable := _LoadExternal);
END_IF
END_METHOD

(*!
<summary>Checks workflow round-trip deserialization, rollback on missing PLC bindings, execution and reset.</summary>
<description>Exercises embedded and external dependencies, activity and condition declarations, and dynamic disposal.
Reports a failed bound load before fixture cleanup and test completion.</description>
<param name="assertions">Valid assertion context borrowed from the active case.</param>
*)
METHOD PRIVATE testLoadConfiguration
VAR_INPUT
	assertions : REFERENCE TO TOF_Testing.Assertions;
END_VAR
VAR
	initialStep : UINT := 3;
	firstLimit : UINT := 4;
	secondLimit : UINT := 8;
	mutated : UINT := 77;
	limits : ARRAY [0..1] OF __SYSTEM.AnyType;
	embeddedTask : POINTER TO WorkflowBindingTask;
	embeddedComparer : POINTER TO WorkflowBindingTask;
	ifElse : TOF_Workflow.IIfElseActivity;
	rootScope : TOF_Workflow.IDeclaredVariableContainer;
	conditionScope : TOF_Workflow.IDeclaredVariableContainer;
	localStep : TOF_Core.GENERIC_VALUE;
	limitElement : TOF_Core.GENERIC_VALUE;
	thresholdElement : TOF_Core.GENERIC_VALUE;
	exceptionCode : __SYSTEM.ExceptionCode;
	exception : TOF_Core.IException;
	configurationError : TOF_Workflow.IWorkflowConfigurationException;
	caught : BOOL;
	ready : BOOL;
	i : DINT;
END_VAR
_LoadSource.DeclareVariable(name := 'Step', initialValue := initialStep);
_LoadSource.BindPlcVariable(name := 'External', plcVariable := _LoadExternal);
limits[0] := TOF_Workflow.Workflows.GetValueDescriptor(value := firstLimit);
limits[1] := TOF_Workflow.Workflows.GetValueDescriptor(value := secondLimit);
_LoadIf.DeclareArray(name := 'Limits', initialValues := ADR(limits[0]), elementCount := 2);
_LoadIf.DeclareVariable(name := 'LocalStep', initialValue := initialStep);

_LoadCompare.DeclareVariable(name := 'Threshold', initialValue := initialStep);
_LoadCompare.ConfigureVariable(
	firstVariableName := 'LocalStep',
	comparisonOperator := TOF_Workflow.COMPARISON_OPERATOR.EQUAL,
	secondVariableName := 'Threshold'
);
embeddedComparer := __NEW(WorkflowBindingTask(name := "Embedded comparer"));

IF embeddedComparer = 0 THEN
	TOF_Core.DynamicMemoryManager.RaiseAllocationFailure();
END_IF

_LoadCompare.ConfigureEmbeddedComparer(comparer := embeddedComparer^);
embeddedTask := __NEW(WorkflowBindingTask(name := "Embedded task"));

IF embeddedTask = 0 THEN
	TOF_Core.DynamicMemoryManager.RaiseAllocationFailure();
END_IF

_LoadEmbeddedInvoke.ConfigureEmbeddedTask(task := embeddedTask^);
_LoadExternalInvoke.ConfigureExternalTask(task := _BindingExternal, key := 'axis');
_LoadAssign.ConfigureFromVariable(targetVariableName := 'LocalStep', sourceVariableName := 'External');

_LoadSequence.AddChildActivity(activity := _LoadEmbeddedInvoke);
_LoadSequence.AddChildActivity(activity := _LoadExternalInvoke);
_LoadSequence.AddChildActivity(activity := _LoadAssign);
_LoadIf.Configure(condition := _LoadCompare, trueActivity := _LoadSequence, falseActivity := 0);
_LoadSource.SetRootActivity(rootActivity := _LoadIf);

_ConfigWriter.Serialize(source := _LoadSource, document := _ConfigDocument);
_BindLoadVariables := FALSE;

__TRY
	_Loaded := _LoadLoader.Load(
		reader := _LoadReader,
		root := _LoadReader.Parse(document := _ConfigDocument),
		factory := THIS^,
		dependencyFactory := THIS^,
		resolver := THIS^,
		binder := THIS^
	);
__CATCH(exceptionCode)
	exception := TOF_Core.ExceptionManager.GetLastException(
		exceptionCode := exceptionCode,
		catchPointNamespaceName := NamespaceName,
		catchPointPOUName := __POUNAME(),
		catchPointPosition := __POSITION()
	);
	caught := exception <> 0 AND_THEN __QUERYINTERFACE(exception, configurationError);
__ENDTRY

IF NOT caught AND_THEN exception <> 0 THEN
	assertions.ThatBool(
		actual := FALSE,
		message := TO_WSTRING(TOF_Core.Strings.Concat255('Unbound workflow load: ', TO_STRING(exception.GetMessage())))
	).IsTrue();
ELSE
	assertions.ThatBool(
		actual := caught AND_THEN _Loaded = 0,
		message := "Unresolved required PLC variable must abort and roll back load"
	).IsTrue();
END_IF

IF _Loaded <> 0 THEN
	assertions.ThatBool(
		actual := TryReleaseLoadedWorkflow(),
		message := "Release any unexpected workflow after the unbound load"
	).IsTrue();
END_IF

TOF_Core.DynamicMemoryManager.RaiseIfAllocationFailed();

_BindLoadVariables := TRUE;
_LoadExternal := 11;
caught := FALSE;
__TRY
	_Loaded := _LoadLoader.Load(
		reader := _LoadReader,
		root := _LoadReader.Parse(document := _ConfigDocument),
		factory := THIS^,
		dependencyFactory := THIS^,
		resolver := THIS^,
		binder := THIS^
	);
__CATCH(exceptionCode)
	caught := TRUE;
	exception := TOF_Core.ExceptionManager.GetLastException(
		exceptionCode := exceptionCode,
		catchPointNamespaceName := NamespaceName,
		catchPointPOUName := __POUNAME(),
		catchPointPosition := __POSITION()
	);

	IF exception <> 0 THEN
		assertions.ThatBool(
			actual := FALSE,
			message := TO_WSTRING(TOF_Core.Strings.Concat255('Bound workflow load: ', TO_STRING(exception.GetMessage())))
		).IsTrue();
	ELSE
		assertions.ThatBool(
			actual := FALSE,
			message := TO_WSTRING(TOF_Core.Strings.Concat255('Bound workflow load raised PLC exception ', TO_STRING(exceptionCode)))
		).IsTrue();
	END_IF
__ENDTRY

IF NOT caught THEN
	assertions.ThatBool(
		actual := _Loaded <> 0 AND_THEN _Loaded.State = TOF_Workflow.WORKFLOW_ELEMENT_STATE.PASSIVE_READY,
		message := "Loaded workflow must be ready without auto-starting"
	).IsTrue();
END_IF

IF _Loaded <> 0 THEN
	_Loaded.RequestStart();

	FOR i := 1 TO 6 DO
		IF _Loaded.Busy THEN
			_Loaded.Execute();
		END_IF
	END_FOR

	assertions.ThatBool(
		actual := _Loaded.State = TOF_Workflow.WORKFLOW_ELEMENT_STATE.PASSIVE_COMPLETED,
		message := "Loaded workflow must execute embedded and external tasks and branch assignment"
	).IsTrue();

	ready := __QUERYINTERFACE(_Loaded.RootActivity, ifElse)
		AND_THEN __QUERYINTERFACE(_Loaded.RootActivity, rootScope)
		AND_THEN __QUERYINTERFACE(ifElse.Condition, conditionScope);
	assertions.ThatBool(
		actual := ready,
		message := "Loaded root and condition must expose declaration containers"
	).IsTrue();

	IF ready THEN
		localStep := rootScope.GetDeclaredElement(name := 'LocalStep', index := 0);
		limitElement := rootScope.GetDeclaredElement(name := 'Limits', index := 1);
		thresholdElement := conditionScope.GetDeclaredElement(name := 'Threshold', index := 0);
		assertions.ThatBool(
			actual := localStep.AsUInt() = 11 AND_THEN limitElement.AsUInt() = 8 AND_THEN thresholdElement.AsUInt() = 3,
			message := "Loaded execution must update target declaration and preserve array and condition values"
		).IsTrue();

		limitElement.ChangeValueByAny(value := mutated);
		thresholdElement.ChangeValueByAny(value := mutated);
		_Loaded.RequestReset();

		assertions.ThatBool(
			actual := _Loaded.State = TOF_Workflow.WORKFLOW_ELEMENT_STATE.PASSIVE_READY
				AND_THEN localStep.AsUInt() = 3
				AND_THEN limitElement.AsUInt() = 8
				AND_THEN thresholdElement.AsUInt() = 3,
			message := "Resetting a loaded workflow must restore activity and condition declarations in place"
		).IsTrue();
	END_IF

	assertions.ThatBool(
		actual := TryReleaseLoadedWorkflow(),
		message := "Release the dynamically loaded workflow"
	).IsTrue();
END_IF

_LoadSource.DisposeDynamicChildren();
TOF_Core.DynamicMemoryManager.RaiseIfAllocationFailed();
END_METHOD

(*!
<summary>Verifies that workflow element deserialization rejects null context and context-free succeeds.</summary>
<description>
A workflow element requiring a loader raises WorkflowConfiguration when deserialized with context = 0.
A context-free element (DelayActivity) succeeds when deserialized with context = 0.
</description>
<param name="assertions">Valid assertion context borrowed from the active case.</param>
*)
METHOD PRIVATE testDeserializeNullContextRejection
VAR_INPUT
	assertions : REFERENCE TO TOF_Testing.Assertions;
END_VAR
VAR
	workflowNode : TOF_Core.CONFIGURATION_NODE;
	delayNode : TOF_Core.CONFIGURATION_NODE;
	caught : BOOL;
	exceptionCode : __SYSTEM.ExceptionCode;
	exception : TOF_Core.IException;
	configurationError : TOF_Workflow.IWorkflowConfigurationException;
END_VAR
_ConfigWriter.Serialize(source := _NullContextSequence, document := _ConfigDocument);
workflowNode := _LoadReader.Parse(document := _ConfigDocument);

caught := FALSE;
__TRY
	_NullContextSequence.Deserialize(reader := _LoadReader, node := workflowNode, context := 0);
__CATCH(exceptionCode)
	exception := TOF_Core.ExceptionManager.GetLastException(
		exceptionCode := exceptionCode,
		catchPointNamespaceName := NamespaceName,
		catchPointPOUName := __POUNAME(),
		catchPointPosition := __POSITION()
	);
	caught := __QUERYINTERFACE(exception, configurationError);
__ENDTRY

assertions.ThatBool(
	actual := caught,
	message := "Workflow element requiring loader must reject null deserialization context"
).IsTrue();

_NullContextDelay.Interval := T#5S;
_ConfigWriter.Serialize(source := _NullContextDelay, document := _ConfigDocument);
delayNode := _LoadReader.Parse(document := _ConfigDocument);

caught := FALSE;
__TRY
	_NullContextDelay.Deserialize(reader := _LoadReader, node := delayNode, context := 0);
__CATCH(exceptionCode)
	caught := TRUE;
__ENDTRY

assertions.ThatBool(
	actual := caught,
	message := "Context-free workflow element must succeed with null deserialization context"
).IsFalse();
assertions.ThatTime(
	actual := _NullContextDelay.Interval,
	message := "Delay interval must be restored"
).ToBe(expected := T#5S);

TOF_Core.DynamicMemoryManager.RaiseIfAllocationFailed();
END_METHOD

(*!
<summary>Verifies formatting and parsing of logical and comparison operators.</summary>
<param name="assertions">Valid assertion context borrowed from the active case.</param>
*)
METHOD PRIVATE testOperatorSerialization
VAR_INPUT
	assertions : REFERENCE TO TOF_Testing.Assertions;
END_VAR
VAR
	caught : BOOL;
	exceptionCode : __SYSTEM.ExceptionCode;
	exception : TOF_Core.IException;
	configurationError : TOF_Workflow.IWorkflowConfigurationException;
	parsedComp : TOF_Workflow.COMPARISON_OPERATOR;
	parsedLog : TOF_Workflow.LOGICAL_OPERATOR;
END_VAR
// Format comparison operators
assertions.ThatString(
	actual := TOF_Workflow.Workflows.FormatComparisonOperator(comparisonOperator := TOF_Workflow.COMPARISON_OPERATOR.EQUAL),
	message := "Format EQUAL"
).ToBe(expected := '=');
assertions.ThatString(
	actual := TOF_Workflow.Workflows.FormatComparisonOperator(comparisonOperator := TOF_Workflow.COMPARISON_OPERATOR.NOT_EQUAL),
	message := "Format NOT_EQUAL"
).ToBe(expected := '<>');
assertions.ThatString(
	actual := TOF_Workflow.Workflows.FormatComparisonOperator(comparisonOperator := TOF_Workflow.COMPARISON_OPERATOR.LESS_THAN),
	message := "Format LESS_THAN"
).ToBe(expected := '<');
assertions.ThatString(
	actual := TOF_Workflow.Workflows.FormatComparisonOperator(comparisonOperator := TOF_Workflow.COMPARISON_OPERATOR.LESS_THAN_OR_EQUAL),
	message := "Format LESS_THAN_OR_EQUAL"
).ToBe(expected := '<=');
assertions.ThatString(
	actual := TOF_Workflow.Workflows.FormatComparisonOperator(comparisonOperator := TOF_Workflow.COMPARISON_OPERATOR.GREATER_THAN),
	message := "Format GREATER_THAN"
).ToBe(expected := '>');
assertions.ThatString(
	actual := TOF_Workflow.Workflows.FormatComparisonOperator(comparisonOperator := TOF_Workflow.COMPARISON_OPERATOR.GREATER_THAN_OR_EQUAL),
	message := "Format GREATER_THAN_OR_EQUAL"
).ToBe(expected := '>=');

// Parse comparison operators and synonyms
parsedComp := TOF_Workflow.Workflows.ParseComparisonOperator(rawOperator := '=');
assertions.ThatBool(actual := parsedComp = TOF_Workflow.COMPARISON_OPERATOR.EQUAL, message := "Parse =").IsTrue();

parsedComp := TOF_Workflow.Workflows.ParseComparisonOperator(rawOperator := '==');
assertions.ThatBool(actual := parsedComp = TOF_Workflow.COMPARISON_OPERATOR.EQUAL, message := "Parse ==").IsTrue();

parsedComp := TOF_Workflow.Workflows.ParseComparisonOperator(rawOperator := '<>');
assertions.ThatBool(
	actual := parsedComp = TOF_Workflow.COMPARISON_OPERATOR.NOT_EQUAL,
	message := "Parse <>"
).IsTrue();

parsedComp := TOF_Workflow.Workflows.ParseComparisonOperator(rawOperator := '!=');
assertions.ThatBool(
	actual := parsedComp = TOF_Workflow.COMPARISON_OPERATOR.NOT_EQUAL,
	message := "Parse !="
).IsTrue();

parsedComp := TOF_Workflow.Workflows.ParseComparisonOperator(rawOperator := '<');
assertions.ThatBool(
	actual := parsedComp = TOF_Workflow.COMPARISON_OPERATOR.LESS_THAN,
	message := "Parse <"
).IsTrue();

parsedComp := TOF_Workflow.Workflows.ParseComparisonOperator(rawOperator := '<=');
assertions.ThatBool(
	actual := parsedComp = TOF_Workflow.COMPARISON_OPERATOR.LESS_THAN_OR_EQUAL,
	message := "Parse <="
).IsTrue();

parsedComp := TOF_Workflow.Workflows.ParseComparisonOperator(rawOperator := '>');
assertions.ThatBool(
	actual := parsedComp = TOF_Workflow.COMPARISON_OPERATOR.GREATER_THAN,
	message := "Parse >"
).IsTrue();

parsedComp := TOF_Workflow.Workflows.ParseComparisonOperator(rawOperator := '>=');
assertions.ThatBool(
	actual := parsedComp = TOF_Workflow.COMPARISON_OPERATOR.GREATER_THAN_OR_EQUAL,
	message := "Parse >="
).IsTrue();

// Invalid comparison operator
caught := FALSE;
__TRY
	parsedComp := TOF_Workflow.Workflows.ParseComparisonOperator(rawOperator := 'INVALID');
__CATCH(exceptionCode)
	exception := TOF_Core.ExceptionManager.GetLastException(
		exceptionCode := exceptionCode,
		catchPointNamespaceName := NamespaceName,
		catchPointPOUName := __POUNAME(),
		catchPointPosition := __POSITION()
	);
	caught := __QUERYINTERFACE(exception, configurationError);
__ENDTRY
assertions.ThatBool(actual := caught, message := "Unknown comparison operator must raise").IsTrue();

// Format logical operators
assertions.ThatString(
	actual := TOF_Workflow.Workflows.FormatLogicalOperator(logicalOperator := TOF_Workflow.LOGICAL_OPERATOR.AND_),
	message := "Format AND_"
).ToBe(expected := 'AND');
assertions.ThatString(
	actual := TOF_Workflow.Workflows.FormatLogicalOperator(logicalOperator := TOF_Workflow.LOGICAL_OPERATOR.OR_),
	message := "Format OR_"
).ToBe(expected := 'OR');

// Parse logical operators
parsedLog := TOF_Workflow.Workflows.ParseLogicalOperator(rawOperator := 'AND');
assertions.ThatBool(actual := parsedLog = TOF_Workflow.LOGICAL_OPERATOR.AND_, message := "Parse AND").IsTrue();

parsedLog := TOF_Workflow.Workflows.ParseLogicalOperator(rawOperator := 'and');
assertions.ThatBool(
	actual := parsedLog = TOF_Workflow.LOGICAL_OPERATOR.AND_,
	message := "Parse and lowercase"
).IsTrue();

parsedLog := TOF_Workflow.Workflows.ParseLogicalOperator(rawOperator := 'AND_');
assertions.ThatBool(actual := parsedLog = TOF_Workflow.LOGICAL_OPERATOR.AND_, message := "Parse AND_").IsTrue();

parsedLog := TOF_Workflow.Workflows.ParseLogicalOperator(rawOperator := 'OR');
assertions.ThatBool(actual := parsedLog = TOF_Workflow.LOGICAL_OPERATOR.OR_, message := "Parse OR").IsTrue();

parsedLog := TOF_Workflow.Workflows.ParseLogicalOperator(rawOperator := 'or');
assertions.ThatBool(
	actual := parsedLog = TOF_Workflow.LOGICAL_OPERATOR.OR_,
	message := "Parse or lowercase"
).IsTrue();

parsedLog := TOF_Workflow.Workflows.ParseLogicalOperator(rawOperator := 'OR_');
assertions.ThatBool(actual := parsedLog = TOF_Workflow.LOGICAL_OPERATOR.OR_, message := "Parse OR_").IsTrue();

// Invalid logical operator
caught := FALSE;
__TRY
	parsedLog := TOF_Workflow.Workflows.ParseLogicalOperator(rawOperator := 'XOR');
__CATCH(exceptionCode)
	exception := TOF_Core.ExceptionManager.GetLastException(
		exceptionCode := exceptionCode,
		catchPointNamespaceName := NamespaceName,
		catchPointPOUName := __POUNAME(),
		catchPointPosition := __POSITION()
	);
	caught := __QUERYINTERFACE(exception, configurationError);
__ENDTRY
assertions.ThatBool(actual := caught, message := "Unknown logical operator must raise").IsTrue();

TOF_Core.DynamicMemoryManager.RaiseIfAllocationFailed();
END_METHOD

(*!
<summary>Attempts to release the owned result of a configuration load.</summary>
<description>Clears the stored alias before release. Succeeds if no workflow is owned.</description>
*)
METHOD TryReleaseLoadedWorkflow : BOOL
VAR
	instance : TOF_Core.IObject;
END_VAR
IF _Loaded = 0 THEN
	TryReleaseLoadedWorkflow := TRUE;

	RETURN;
END_IF

instance := _Loaded;
_Loaded := 0;
TryReleaseLoadedWorkflow := TOF_Core.Memory.TryReleaseDynamicObject(instance := instance);
END_METHOD

(*!
<summary>Clears a still-owned loaded workflow if the fixture is unloaded before case teardown.</summary>
<param name="bInCopyCode">TwinCAT copy-code exit marker. Leave copied ownership with the new instance.</param>
*)
METHOD FB_exit : BOOL
VAR_INPUT
	bInCopyCode : BOOL;
END_VAR
IF NOT bInCopyCode THEN
	TryReleaseLoadedWorkflow();
END_IF

FB_exit := TRUE;
END_METHOD

END_FUNCTION_BLOCK

// ---- Tests/Workflow/WorkflowBindingTask.TcPOU
(*
SPDX-FileCopyrightText: © 2026 Oleksandr Tiutyk <trofimich@gmail.com>
SPDX-License-Identifier: MIT
License: https://opensource.org/license/mit
*)

(*!
<summary>Exercises task and comparer bindings on the same concrete instance.</summary>
<description>Both interfaces expose this object to the ownership registry.</description>
*)

{attribute 'no_explicit_call' := 'do not call this function block directly'}
{attribute 'enable_dynamic_creation'}
FUNCTION_BLOCK WorkflowBindingTask EXTENDS TOF_Tasks.Task
IMPLEMENTS TOF_Core.IComparer, TOF_Core.IConfigurationSerializable
VAR_STAT
	_ClassName : STRING := __POUNAME();
END_VAR

(*!
<summary>Returns the initialized static name of this concrete fixture.</summary>
*)
{attribute 'monitoring' := 'call'}
PROPERTY ClassName : REFERENCE TO STRING
GET
ClassName REF= _ClassName;
END_GET
END_PROPERTY

(*!
<summary>Borrows the test project namespace without changing it.</summary>
*)
{attribute 'monitoring' := 'call'}
PROPERTY NamespaceName : REFERENCE TO STRING
GET
NamespaceName REF= CurrentNamespace.Name;
END_GET
END_PROPERTY

(*!
<summary>Reports the size of this concrete fixture in bytes.</summary>
*)
{attribute 'monitoring' := 'call'}
PROPERTY SelfSize : ULINT
GET
SelfSize := XSIZEOF(THIS^);
END_GET
END_PROPERTY

(*!
<summary>Completes immediately.</summary>
<description>This fixture does not use resources.</description>
*)
METHOD PROTECTED OnRunning
VAR_OUTPUT
	processingState : TOF_Tasks.TASK_PROCESSING_STATE;
END_VAR
VAR_IN_OUT
	stopReasonMessage : TOF_Core.ERROR_MESSAGE;
END_VAR
processingState := TOF_Tasks.TASK_PROCESSING_STATE.DONE;
END_METHOD

(*!
<summary>Compares test operands by their natural ordering.</summary>
<description>Borrows both operands for this call.</description>
*)
METHOD Compare : TOF_Core.COMPARISON_RESULT
VAR_INPUT
	first : TOF_Core.GENERIC_VALUE;
	second : TOF_Core.GENERIC_VALUE;
END_VAR
Compare := first.CompareTo(otherValue := second);
END_METHOD

(*!
<summary>Writes the configuration fields for this object.</summary>
<description>Borrows the writer for this call. A failure invalidates the current output document.</description>
*)
METHOD Serialize
VAR_INPUT
	writer : TOF_Core.IConfigurationWriter;
END_VAR
VAR
	displayName : WSTRING;
END_VAR
displayName := Name;
writer.WriteValue(
	name := 'name',
	valueType := TOF_Core.CONFIGURATION_VALUE_TYPE.TYPE_WSTRING,
	data := ADR(displayName),
	size := SIZEOF(displayName)
);
END_METHOD

(*!
<summary>Restores this fresh instance from its configuration object.</summary>
<description>
The reader and document node are borrowed for this call. The deserialization context is ignored.
On failure discard the partial instance.
</description>
<param name="reader">Active configuration reader.</param>
<param name="node">Object node to read fields from.</param>
<param name="context">Configuration deserialization context; ignored by this task.</param>
*)
METHOD Deserialize
VAR_INPUT
	reader : TOF_Core.IConfigurationReader;
	node : TOF_Core.CONFIGURATION_NODE;
	context : TOF_Core.IConfigurationDeserializationContext;
END_VAR
VAR
	displayName : WSTRING;
END_VAR
reader.ReadValue(
	node := reader.GetField(node := node, name := 'name'),
	valueType := TOF_Core.CONFIGURATION_VALUE_TYPE.TYPE_WSTRING,
	data := ADR(displayName),
	size := SIZEOF(displayName)
);
Name := displayName;
END_METHOD

END_FUNCTION_BLOCK

// ---- Tests/Workflow/WorkflowContractActivity.TcPOU
(*
SPDX-FileCopyrightText: © 2026 Oleksandr Tiutyk <trofimich@gmail.com>
SPDX-License-Identifier: MIT
License: https://opensource.org/license/mit
*)

(*!
<summary>Provides controlled execution and formatter failures for workflow contract tests.</summary>
<description>
Persistent test instances own their borrowed configuration and exception template. No hardware effects or
terminal allocation injection are performed. The fixture can defer its initial resetting step. All observations are task-local.
</description>
*)

{attribute 'enable_dynamic_creation'}
{attribute 'no_explicit_call' := 'do not call this function block directly'}
{attribute 'no_assign'}
FUNCTION_BLOCK WorkflowContractActivity EXTENDS TOF_Workflow.Activity
VAR_INPUT
	//! <summary>Raises an ordinary work exception on every running call while enabled.</summary>
	throwOrdinaryFailure : BOOL;
	//! <summary>Raises a concrete exception whose message formatter itself raises.</summary>
	throwMessageFailure : BOOL;
	//! <summary>Completes running immediately when no injected failure is enabled.</summary>
	completeRunning : BOOL;
	//! <summary>Keeps the first reset step pending until the next Execute call.</summary>
	deferFirstResetStep : BOOL;
	//! <summary>Optional persistent observer incremented on ordinary destruction of a factory fixture.</summary>
	exitCount : REFERENCE TO DINT;
END_VAR
VAR_OUTPUT
	//! <summary>Number of fresh or resumed start callbacks.</summary>
	startCount : DINT;
	//! <summary>Number of running callbacks, including entry calls.</summary>
	runningCount : DINT;
	//! <summary>Number of stopping callbacks.</summary>
	stopCount : DINT;
END_VAR
VAR_STAT
	//! <summary>Initialized static metadata available during inherited base initialization.</summary>
	_ClassName : STRING := __POUNAME();
END_VAR
VAR
	_MessageFailure : ThrowingGetMessageException;
END_VAR

(*!
<summary>Returns the initialized static name of this concrete fixture.</summary>
*)
{attribute 'monitoring' := 'call'}
PROPERTY ClassName : REFERENCE TO STRING
GET
ClassName REF= _ClassName;
END_GET
END_PROPERTY

(*!
<summary>Borrows the test project namespace without changing it.</summary>
*)
{attribute 'monitoring' := 'call'}
PROPERTY NamespaceName : REFERENCE TO STRING
GET
NamespaceName REF= CurrentNamespace.Name;
END_GET
END_PROPERTY

(*!
<summary>Reports the size of this concrete fixture in bytes.</summary>
*)
{attribute 'monitoring' := 'call'}
PROPERTY SelfSize : ULINT
GET
SelfSize := XSIZEOF(THIS^);
END_GET
END_PROPERTY

(*!
<summary>Counts execution and produces the selected ordinary result or exception.</summary>
<param name="startRunning">Marks a fresh start for the entry counter.</param>
<param name="startResuming">Marks a resumed start for the entry counter.</param>
<param name="haltReason">Unused because this probe does not halt.</param>
*)
METHOD PROTECTED OnRunning : TOF_Workflow.ACTIVITY_RUNNING_STATE
VAR_INPUT
	startRunning : BOOL;
	startResuming : BOOL;
END_VAR
VAR_OUTPUT
	haltReason : WSTRING(255);
END_VAR
runningCount := runningCount + 1;

IF startRunning OR_ELSE startResuming THEN
	startCount := startCount + 1;
END_IF

IF throwMessageFailure THEN
	_MessageFailure.Throw(
		sourceNamespaceName := NamespaceName,
		sourceClassName := ClassName,
		sourcePOUName := __POUNAME(),
		sourcePosition := __POSITION(),
		message := "Controlled original workflow failure"
	);
END_IF

IF throwOrdinaryFailure THEN
	TOF_Core.Exceptions.ThrowStandard(
		sourceNamespaceName := NamespaceName,
		sourceClassName := ClassName,
		sourcePOUName := __POUNAME(),
		sourcePosition := __POSITION(),
		message := "Controlled workflow work failure"
	);
END_IF

IF completeRunning THEN
	OnRunning := TOF_Workflow.ACTIVITY_RUNNING_STATE.WORK_COMPLETED;
END_IF
END_METHOD

(*!
<summary>Counts a cooperative stopping step and finishes it immediately.</summary>
<param name="startCancelling">Unused cancellation-entry marker; stopping is immediate.</param>
<param name="startSuspending">Unused suspension-entry marker; stopping is immediate.</param>
<param name="haltReason">Unused because this probe does not halt.</param>
*)
METHOD PROTECTED OnStopping : TOF_Workflow.ACTIVITY_STOPPING_STATE
VAR_INPUT
	startCancelling : BOOL;
	startSuspending : BOOL;
END_VAR
VAR_OUTPUT
	haltReason : WSTRING(255);
END_VAR
stopCount := stopCount + 1;

OnStopping := TOF_Workflow.ACTIVITY_STOPPING_STATE.WORK_STOPPED;
END_METHOD

(*!
<summary>Optionally defers reset completion by one step.</summary>
<param name="startResetting">TRUE only on entry to reset.</param>
*)
METHOD PROTECTED OnResetting : TOF_Workflow.ACTIVITY_RESETTING_STATE
VAR_INPUT
	startResetting : BOOL;
END_VAR
IF startResetting AND_THEN deferFirstResetStep THEN
	OnResetting := TOF_Workflow.ACTIVITY_RESETTING_STATE.WORK_IN_PROGRESS;
ELSE
	OnResetting := TOF_Workflow.ACTIVITY_RESETTING_STATE.WORK_RESET;
END_IF
END_METHOD

(*!
<summary>Reports ordinary destruction to an optional persistent counter.</summary>
<description>The suite keeps the counter alive until disposal. Counting a callback does not certify physical deallocation.</description>
<param name="bInCopyCode">TwinCAT online-change indicator.</param>
*)
METHOD FB_exit : BOOL
VAR_INPUT
	bInCopyCode : BOOL;
END_VAR
IF NOT bInCopyCode AND_THEN __ISVALIDREF(exitCount) THEN
	exitCount := exitCount + 1;
END_IF
END_METHOD

END_FUNCTION_BLOCK

// ---- Tests/Workflow/WorkflowContractWorkflow.TcPOU
(*
SPDX-FileCopyrightText: © 2026 Oleksandr Tiutyk <trofimich@gmail.com>
SPDX-License-Identifier: MIT
License: https://opensource.org/license/mit
*)

(*!
<summary>Observes workflow hooks and injects one recoverable initialization failure.</summary>
<description>
Variable storage belongs to this persistent fixture. The initialization failure is raised only after one
ordinary binding was added, allowing the caller to observe the configured retry policy.
</description>
*)

{attribute 'no_explicit_call' := 'do not call this function block directly'}
{attribute 'no_assign'}
FUNCTION_BLOCK WorkflowContractWorkflow EXTENDS TOF_Workflow.Workflow
VAR_INPUT
	//! <summary>Raises once after registering the initialization binding.</summary>
	throwInitialization : BOOL;
END_VAR
VAR_OUTPUT
	//! <summary>Total calls to InitializeVariables.</summary>
	initializationCount : DINT;
	//! <summary>Total calls to OnAfterRootActivityExecute.</summary>
	afterCount : DINT;
END_VAR
VAR_STAT
	//! <summary>Distinct static field to avoid redeclaring inherited Workflow metadata.</summary>
	_ProbeClassName : STRING := __POUNAME();
END_VAR
VAR
	_RegisteredValue : DINT;
END_VAR

(*!
<summary>Returns the initialized static name of this concrete fixture.</summary>
*)
{attribute 'monitoring' := 'call'}
PROPERTY ClassName : REFERENCE TO STRING
GET
ClassName REF= _ProbeClassName;
END_GET
END_PROPERTY

(*!
<summary>Borrows the test project namespace without changing it.</summary>
*)
{attribute 'monitoring' := 'call'}
PROPERTY NamespaceName : REFERENCE TO STRING
GET
// SA0006: Read-only namespace string borrowed across test tasks.
{analysis -6}
NamespaceName REF= CurrentNamespace.Name;
{analysis +6}
END_GET
END_PROPERTY

(*!
<summary>Reports the size of this concrete fixture in bytes.</summary>
*)
{attribute 'monitoring' := 'call'}
PROPERTY SelfSize : ULINT
GET
SelfSize := XSIZEOF(THIS^);
END_GET
END_PROPERTY

(*!
<summary>Registers persistent fixture storage and optionally interrupts the first attempt.</summary>
*)
METHOD PROTECTED InitializeVariables
initializationCount := initializationCount + 1;
BindPlcVariable(name := 'Initialized', plcVariable := _RegisteredValue);

IF throwInitialization THEN
	throwInitialization := FALSE;

	TOF_Core.Exceptions.ThrowStandard(
		sourceNamespaceName := NamespaceName,
		sourceClassName := ClassName,
		sourcePOUName := __POUNAME(),
		sourcePosition := __POSITION(),
		message := "Controlled variable initialization failure"
	);
END_IF
END_METHOD

(*!
<summary>Counts completion of the workflow execution boundary.</summary>
*)
METHOD PROTECTED OnAfterRootActivityExecute
afterCount := afterCount + 1;
END_METHOD

END_FUNCTION_BLOCK

// ---- Tests/Workflow/WorkflowContractTask.TcPOU
(*
SPDX-FileCopyrightText: © 2026 Oleksandr Tiutyk <trofimich@gmail.com>
SPDX-License-Identifier: MIT
License: https://opensource.org/license/mit
*)

(*!
<summary>Provides controlled processing and delayed stopping for the workflow task adapter.</summary>
<description>
The test owns this task and any injected resource manager. Cancel with an injected manager only after
acquisition completes. No native I/O or terminal allocation injection is performed. Observations are task-local.
</description>
*)

{attribute 'no_explicit_call' := 'do not call this function block directly'}
{attribute 'no_assign'}
FUNCTION_BLOCK WorkflowContractTask EXTENDS TOF_Tasks.Task
VAR_INPUT
	//! <summary>Result returned by each processing callback.</summary>
	processingResult : TOF_Tasks.TASK_PROCESSING_STATE;
	//! <summary>Number of stopping callbacks required before resource release.</summary>
	requiredStopCalls : DINT := 1;
	//! <summary>Optional persistent synthetic resource manager; stable until task stopping completes.</summary>
	resource : TOF_Core.IResourceManager;
END_VAR
VAR_OUTPUT
	//! <summary>Number of processing callbacks since reset.</summary>
	processingCount : DINT;
	//! <summary>Number of stopping callbacks since reset.</summary>
	stopCount : DINT;
END_VAR
VAR_STAT
	//! <summary>Initialized static metadata available during inherited base initialization.</summary>
	_ClassName : STRING := __POUNAME();
END_VAR

(*!
<summary>Returns the initialized static name of this concrete fixture.</summary>
*)
{attribute 'monitoring' := 'call'}
PROPERTY ClassName : REFERENCE TO STRING
GET
ClassName REF= _ClassName;
END_GET
END_PROPERTY

(*!
<summary>Borrows the test project namespace without changing it.</summary>
*)
{attribute 'monitoring' := 'call'}
PROPERTY NamespaceName : REFERENCE TO STRING
GET
NamespaceName REF= CurrentNamespace.Name;
END_GET
END_PROPERTY

(*!
<summary>Reports the size of this concrete fixture in bytes.</summary>
*)
{attribute 'monitoring' := 'call'}
PROPERTY SelfSize : ULINT
GET
SelfSize := XSIZEOF(THIS^);
END_GET
END_PROPERTY

(*!
<summary>Returns the optional synthetic resource borrowed by this test task.</summary>
*)
PROPERTY ResourceManager : TOF_Core.IResourceManager
GET
ResourceManager := resource;
END_GET
END_PROPERTY

(*!
<summary>Records a processing callback and returns its configured outcome.</summary>
<param name="processingState">Receives the configured synthetic outcome.</param>
<param name="stopReasonMessage">Receives the synthetic failure or internal-abort diagnostic.</param>
*)
METHOD PROTECTED OnRunning
VAR_OUTPUT
	processingState : TOF_Tasks.TASK_PROCESSING_STATE;
END_VAR
VAR_IN_OUT
	stopReasonMessage : TOF_Core.ERROR_MESSAGE;
END_VAR
processingCount := processingCount + 1;
processingState := processingResult;

IF processingResult = TOF_Tasks.TASK_PROCESSING_STATE.ERROR THEN
	stopReasonMessage := "Controlled task processing failure";
ELSIF processingResult = TOF_Tasks.TASK_PROCESSING_STATE.ABORTED THEN
	stopReasonMessage := "Controlled task internal abort";
END_IF
END_METHOD

(*!
<summary>Waits for the configured number of stopping callbacks without repeating work.</summary>
<param name="readyToRelease">Combines inherited readiness with the configured synthetic stopping delay.</param>
*)
METHOD PROTECTED OnStopping
VAR_OUTPUT
	readyToRelease : BOOL;
END_VAR
VAR
	baseReady : BOOL;
END_VAR
SUPER^.OnStopping(readyToRelease => baseReady);

stopCount := stopCount + 1;
readyToRelease := baseReady AND_THEN stopCount >= requiredStopCalls;
END_METHOD

(*!
<summary>Clears per-run counters while preserving the configured failure and resource inputs.</summary>
*)
METHOD PROTECTED OnReset
SUPER^.OnReset();

processingCount := 0;
stopCount := 0;
END_METHOD

END_FUNCTION_BLOCK

// ---- Tests/Workflow/WorkflowDelayPauseRemainingTest.TcPOU
(*
SPDX-FileCopyrightText: © 2026 Oleksandr Tiutyk <trofimich@gmail.com>
SPDX-License-Identifier: MIT
License: https://opensource.org/license/mit
*)

(*!
<summary>Checks remaining delay duration across two pauses and after reset.</summary>
<description>
Advances one bounded step per PLC cycle. Uses independent task timestamps and a forty-second deadline.
Each pause exceeds the nominal active duration. Run without debugger pauses or clock adjustments.
The task must sample the two active segments before expiry. Diagnostics include the last sampling gap.
</description>
*)

{attribute 'no_assign'}
{attribute 'no_explicit_call' := 'do not call this function block directly'}
FUNCTION_BLOCK WorkflowDelayPauseRemainingTest EXTENDS TOF_Testing.MultiCycleTest
VAR_STAT
	{attribute 'hide'}
	_ClassName : STRING := __POUNAME();
END_VAR
VAR
	_Phase : DELAY_PAUSE_TEST_PHASE;
	_Delay : TOF_Workflow.DelayActivity(workflow := 0);
	_TestStartedAt : ULINT;
	_SegmentStartedAt : ULINT;
	_PausedAt : ULINT;
	_LastObservedAt : ULINT;
	_ActiveTicks : ULINT;
END_VAR

(*!
<summary>Starts a fresh timing run using the independent task-clock deadline.</summary>
*)
METHOD PROTECTED BeforeTest
_Timeout := T#0S;
_Phase := DELAY_PAUSE_TEST_PHASE.BEFORE_START;
_ActiveTicks := 0;
_LastObservedAt := 0;
END_METHOD

(*!
<summary>Advances one step of suspension, resume, completion or fresh-run timing.</summary>
<description>Completion must fall within the timer quantization and actual observation interval.</description>
*)
METHOD PROTECTED ExecuteTest : TOF_Testing.TEST_CYCLE_RESULT
VAR
	assertions : REFERENCE TO TOF_Testing.Assertions;
	currentTaskTime : ULINT;
	elapsedTicks : ULINT;
	observationGap : ULINT;
END_VAR
VAR CONSTANT
	//! <summary>Active target with room for two observed 740ms scheduling gaps before suspension.</summary>
	interval : TIME := T#5S;
	//! <summary>Active duration observed before each suspension, well below the total interval.</summary>
	beforePause : TIME := T#40MS;
	//! <summary>Suspended duration deliberately exceeding the full interval.</summary>
	pauseDuration : TIME := T#6S;
	//! <summary>Allowance for millisecond quantization over three active segments.</summary>
	tolerance : TIME := T#3MS;
	//! <summary>Independent task-time deadline for reporting a scenario that cannot progress.</summary>
	deadline : TIME := T#40S;
	//! <summary>F_GetTaskTime returns 100ns ticks; TIME is expressed in milliseconds.</summary>
	ticksPerMillisecond : ULINT := 10000;
END_VAR
assertions REF= Assert;
ExecuteTest := TOF_Testing.TEST_CYCLE_RESULT.DONE;

currentTaskTime := Tc2_System.F_GetTaskTime();

IF _Phase <> DELAY_PAUSE_TEST_PHASE.BEFORE_START
	AND_THEN currentTaskTime - _TestStartedAt > TO_ULINT(deadline) * ticksPerMillisecond
THEN
	assertions.ThatBool(actual := FALSE, message := "Delay pause scenario exceeded its independent deadline").IsTrue();

	_Phase := DELAY_PAUSE_TEST_PHASE.FINISHED;

	RETURN;
END_IF

observationGap := currentTaskTime - _LastObservedAt;

CASE _Phase OF
	DELAY_PAUSE_TEST_PHASE.BEFORE_START:
		_TestStartedAt := currentTaskTime;
		_SegmentStartedAt := currentTaskTime;
		_Delay.Interval := interval;
		_Delay.RequestStart();
		_Phase := DELAY_PAUSE_TEST_PHASE.FIRST_RUNNING;

	DELAY_PAUSE_TEST_PHASE.FIRST_RUNNING,
	DELAY_PAUSE_TEST_PHASE.SECOND_RUNNING:
		_Delay.Execute();

		IF _Delay.State <> TOF_Workflow.WORKFLOW_ELEMENT_STATE.ACTIVE_RUNNING THEN
			assertions.ThatBool(
				actual := FALSE,
				message := TO_WSTRING(TOF_Core.Strings.Concat255(
					'Delay before pause: phase=', TO_STRING(_Phase), ', state=', TO_STRING(_Delay.State),
					', segment ms=', TO_STRING((currentTaskTime - _SegmentStartedAt) / ticksPerMillisecond),
					', gap ms=', TO_STRING(observationGap / ticksPerMillisecond),
					', active ms=', TO_STRING(_ActiveTicks / ticksPerMillisecond)
				))
			).IsTrue();
			_Phase := DELAY_PAUSE_TEST_PHASE.FINISHED;

			RETURN;
		END_IF

		IF currentTaskTime - _SegmentStartedAt >= TO_ULINT(beforePause) * ticksPerMillisecond THEN
			_ActiveTicks := _ActiveTicks + currentTaskTime - _SegmentStartedAt;
			_Delay.RequestSuspend();
			assertions.ThatBool(
				actual := _Delay.State = TOF_Workflow.WORKFLOW_ELEMENT_STATE.PASSIVE_SUSPENDED,
				message := "Suspension must stop the timer segment immediately"
			).IsTrue();
			assertions.ThatBool(
				actual := _Delay.Interval = interval,
				message := "Suspension must preserve nominal Interval"
			).IsTrue();
			_PausedAt := currentTaskTime;

			IF _Phase = DELAY_PAUSE_TEST_PHASE.FIRST_RUNNING THEN
				_Phase := DELAY_PAUSE_TEST_PHASE.FIRST_PAUSE;
			ELSE
				_Phase := DELAY_PAUSE_TEST_PHASE.SECOND_PAUSE;
			END_IF
		END_IF

	DELAY_PAUSE_TEST_PHASE.FIRST_PAUSE,
	DELAY_PAUSE_TEST_PHASE.SECOND_PAUSE:
		_Delay.Execute();
		assertions.ThatBool(
			actual := _Delay.State = TOF_Workflow.WORKFLOW_ELEMENT_STATE.PASSIVE_SUSPENDED,
			message := "Executing a suspended delay must not consume the remaining duration"
		).IsTrue();

		IF currentTaskTime - _PausedAt >= TO_ULINT(pauseDuration) * ticksPerMillisecond THEN
			_Delay.RequestStart();
			assertions.ThatBool(
				actual := _Delay.State = TOF_Workflow.WORKFLOW_ELEMENT_STATE.ACTIVE_RUNNING,
				message := "Long suspension must leave a positive active remainder after resume"
			).IsTrue();
			_SegmentStartedAt := currentTaskTime;

			IF _Phase = DELAY_PAUSE_TEST_PHASE.FIRST_PAUSE THEN
				_Phase := DELAY_PAUSE_TEST_PHASE.SECOND_RUNNING;
			ELSE
				_Phase := DELAY_PAUSE_TEST_PHASE.REMAINING_RUNNING;
			END_IF
		END_IF

	DELAY_PAUSE_TEST_PHASE.REMAINING_RUNNING,
	DELAY_PAUSE_TEST_PHASE.FRESH_RUNNING:
		_Delay.Execute();
		elapsedTicks := _ActiveTicks + currentTaskTime - _SegmentStartedAt;

		IF _Delay.State = TOF_Workflow.WORKFLOW_ELEMENT_STATE.PASSIVE_COMPLETED THEN
			assertions.ThatBool(
				actual := elapsedTicks + TO_ULINT(tolerance) * ticksPerMillisecond
					>= TO_ULINT(interval) * ticksPerMillisecond,
				message := "Completion must include the full active interval without suspended wall time"
			).IsTrue();
			assertions.ThatBool(
				actual := elapsedTicks <= TO_ULINT(interval + tolerance) * ticksPerMillisecond + observationGap,
				message := "Completion must retain the active remainder instead of restarting the full interval"
			).IsTrue();
			_Delay.RequestReset();
			assertions.ThatBool(
				actual := _Delay.State = TOF_Workflow.WORKFLOW_ELEMENT_STATE.PASSIVE_READY,
				message := "Reset after completion must prepare a fresh delay"
			).IsTrue();

			IF _Phase = DELAY_PAUSE_TEST_PHASE.REMAINING_RUNNING THEN
				assertions.ThatBool(
					actual := _Delay.Interval = interval,
					message := "Reset must preserve configured Interval"
				).IsTrue();
				_ActiveTicks := 0;
				_SegmentStartedAt := currentTaskTime;
				_Delay.RequestStart();
				assertions.ThatBool(
					actual := _Delay.State = TOF_Workflow.WORKFLOW_ELEMENT_STATE.ACTIVE_RUNNING,
					message := "Fresh start must clear previously accumulated active time"
				).IsTrue();
				_Phase := DELAY_PAUSE_TEST_PHASE.FRESH_RUNNING;
			ELSE
				_Phase := DELAY_PAUSE_TEST_PHASE.FINISHED;
			END_IF
		ELSE
			assertions.ThatBool(
				actual := _Delay.State = TOF_Workflow.WORKFLOW_ELEMENT_STATE.ACTIVE_RUNNING,
				message := "A delay awaiting its remainder must stay RUNNING"
			).IsTrue();
			assertions.ThatBool(
				actual := elapsedTicks <= TO_ULINT(interval + tolerance) * ticksPerMillisecond,
				message := "Delay must complete by the active interval plus timer quantization"
			).IsTrue();
		END_IF
END_CASE

_LastObservedAt := currentTaskTime;

IF _Phase <> DELAY_PAUSE_TEST_PHASE.FINISHED THEN
	ExecuteTest := TOF_Testing.TEST_CYCLE_RESULT.BUSY;
END_IF
END_METHOD

(*!
<summary>Cancels a running or suspended delay and checks that reset leaves it ready.</summary>
<description>DelayActivity uses an in-place timer. Cleanup completes without another PLC cycle.</description>
*)
METHOD PROTECTED AfterTest
IF _Delay.CancellingAllowed THEN
	_Delay.RequestCancel(reason := "Timing scenario teardown");
END_IF

IF _Delay.ResettingAllowed THEN
	_Delay.RequestReset();
END_IF

IF _Delay.State <> TOF_Workflow.WORKFLOW_ELEMENT_STATE.PASSIVE_READY THEN
	IF Outcome = TOF_Testing.TEST_OUTCOME.FAILED THEN
		Tc2_System.ADSLOGSTR(
			msgCtrlMask := Tc2_System.Global_Variables.ADSLOG_MSGTYPE_ERROR,
			msgFmtStr := 'Delay timing fixture did not reset from %s',
			strArg := TO_STRING(_Delay.State)
		);
	ELSE
		RecordFailure(message := "Delay timing fixture did not reset to ready");
	END_IF
END_IF
END_METHOD

(*!
<summary>Borrows the concrete class name. Callers must not modify it.</summary>
*)
{attribute 'monitoring' := 'call'}
PROPERTY ClassName : REFERENCE TO STRING
GET
ClassName REF= _ClassName;
END_GET
END_PROPERTY

(*!
<summary>Borrows the project namespace name. Callers must not modify it.</summary>
*)
{attribute 'monitoring' := 'call'}
PROPERTY NamespaceName : REFERENCE TO STRING
GET
NamespaceName REF= CurrentNamespace.Name;
END_GET
END_PROPERTY

(*!
<summary>Reports the complete instance size in bytes.</summary>
*)
{attribute 'monitoring' := 'call'}
PROPERTY SelfSize : ULINT
GET
SelfSize := XSIZEOF(THIS^);
END_GET
END_PROPERTY

END_FUNCTION_BLOCK

// ---- Tests/Automation/AutomationComponentTestGroup.TcPOU
(*
SPDX-FileCopyrightText: © 2026 Oleksandr Tiutyk <trofimich@gmail.com>
SPDX-License-Identifier: MIT
License: https://opensource.org/license/mit
*)

(*!
<summary>Groups automation lifecycle, policy, event, diagnostics and runner scenarios.</summary>
<description>Owns the fixed case tree and runs its leaves in order in the controller task.</description>
*)

{attribute 'no_assign'}
{attribute 'no_explicit_call' := 'do not call this function block directly'}
FUNCTION_BLOCK AutomationComponentTestGroup EXTENDS TOF_Testing.TestGroup<27>
VAR_STAT
	{attribute 'hide'}
	_ClassName : STRING := __POUNAME();
END_VAR
VAR
	_LifecycleTransitions : AutomationComponentTestCase(
		name := "TestLifecycleTransitions",
		parent := THIS^,
		scenario := AUTOMATION_COMPONENT_TEST_SCENARIO.LIFECYCLE_TRANSITIONS
	);
	_InitializationTimeout : AutomationChildInitializationTimeoutTest(name := "TestInitializationTimeout", parent := THIS^);
	_EnableDisable : AutomationComponentTestCase(
		name := "TestEnableDisable",
		parent := THIS^,
		scenario := AUTOMATION_COMPONENT_TEST_SCENARIO.ENABLE_DISABLE
	);
	_ChildErrorPolicyIgnore : AutomationComponentTestCase(
		name := "TestChildErrorPolicyIgnore",
		parent := THIS^,
		scenario := AUTOMATION_COMPONENT_TEST_SCENARIO.CHILD_ERROR_POLICY_IGNORE
	);
	_ChildErrorPolicySetErrorAndContinue : AutomationComponentTestCase(
		name := "TestChildErrorPolicySetErrorAndContinue",
		parent := THIS^,
		scenario := AUTOMATION_COMPONENT_TEST_SCENARIO.CHILD_ERROR_POLICY_SET_ERROR_AND_CONTINUE
	);
	_ChildErrorPolicySetErrorAndStop : AutomationComponentTestCase(
		name := "TestChildErrorPolicySetErrorAndStop",
		parent := THIS^,
		scenario := AUTOMATION_COMPONENT_TEST_SCENARIO.CHILD_ERROR_POLICY_SET_ERROR_AND_STOP
	);
	_EventBubbling : AutomationComponentTestCase(
		name := "TestEventBubbling",
		parent := THIS^,
		scenario := AUTOMATION_COMPONENT_TEST_SCENARIO.EVENT_BUBBLING
	);
	_EventBubblingStopPropagation : AutomationComponentTestCase(
		name := "TestEventBubblingStopPropagation",
		parent := THIS^,
		scenario := AUTOMATION_COMPONENT_TEST_SCENARIO.EVENT_BUBBLING_STOP_PROPAGATION
	);
	_EventBroadcasting : AutomationComponentTestCase(
		name := "TestEventBroadcasting",
		parent := THIS^,
		scenario := AUTOMATION_COMPONENT_TEST_SCENARIO.EVENT_BROADCASTING
	);
	_InputOutputPhases : AutomationComponentTestCase(
		name := "TestInputOutputPhases",
		parent := THIS^,
		scenario := AUTOMATION_COMPONENT_TEST_SCENARIO.INPUT_OUTPUT_PHASES
	);
	_OutputPhaseStop : AutomationComponentTestCase(
		name := "TestOutputPhaseStop",
		parent := THIS^,
		scenario := AUTOMATION_COMPONENT_TEST_SCENARIO.OUTPUT_PHASE_STOP
	);
	_InputPhaseStop : AutomationComponentTestCase(
		name := "TestInputPhaseStop",
		parent := THIS^,
		scenario := AUTOMATION_COMPONENT_TEST_SCENARIO.INPUT_PHASE_STOP
	);
	_OutputPhaseContinuation : AutomationComponentTestCase(
		name := "TestOutputPhaseContinuation",
		parent := THIS^,
		scenario := AUTOMATION_COMPONENT_TEST_SCENARIO.OUTPUT_PHASE_CONTINUATION
	);
	_PrimaryErrorBeforeLogging : AutomationComponentTestCase(
		name := "TestPrimaryErrorBeforeLogging",
		parent := THIS^,
		scenario := AUTOMATION_COMPONENT_TEST_SCENARIO.PRIMARY_ERROR_BEFORE_LOGGING
	);
	_RunnerHappyPath : AutomationRunnerObservationTest(
		name := "TestRunnerHappyPath",
		parent := THIS^,
		checkInvalidRoots := FALSE
	);
	_RunnerNullComponentGuard : AutomationRunnerObservationTest(
		name := "TestRunnerNullComponentGuard",
		parent := THIS^,
		checkInvalidRoots := TRUE
	);
	_ResetChildPolicies : AutomationComponentTestCase(
		name := "TestResetChildPolicies",
		parent := THIS^,
		scenario := AUTOMATION_COMPONENT_TEST_SCENARIO.RESET_CHILD_POLICIES
	);
	_ResetFromStoppedHook : AutomationComponentTestCase(
		name := "TestResetFromStoppedHook",
		parent := THIS^,
		scenario := AUTOMATION_COMPONENT_TEST_SCENARIO.RESET_FROM_STOPPED_HOOK
	);
	_ParentValidation : AutomationComponentTestCase(
		name := "TestParentValidation",
		parent := THIS^,
		scenario := AUTOMATION_COMPONENT_TEST_SCENARIO.PARENT_VALIDATION
	);
	_DuplicateChild : AutomationComponentTestCase(
		name := "TestDuplicateChild",
		parent := THIS^,
		scenario := AUTOMATION_COMPONENT_TEST_SCENARIO.DUPLICATE_CHILD
	);
	_MismatchedChildParent : AutomationComponentTestCase(
		name := "TestMismatchedChildParent",
		parent := THIS^,
		scenario := AUTOMATION_COMPONENT_TEST_SCENARIO.MISMATCHED_CHILD_PARENT
	);
	_InitializationFailureResult : AutomationComponentTestCase(
		name := "TestInitializationFailureResult",
		parent := THIS^,
		scenario := AUTOMATION_COMPONENT_TEST_SCENARIO.INITIALIZATION_FAILURE_RESULT
	);
	_IndexedLookupContainment : AutomationComponentTestCase(
		name := "TestIndexedLookupContainment",
		parent := THIS^,
		scenario := AUTOMATION_COMPONENT_TEST_SCENARIO.INDEXED_LOOKUP_CONTAINMENT
	);
	_ControllerPluginRecovery : AutomationComponentTestCase(
		name := "TestControllerPluginRecovery",
		parent := THIS^,
		scenario := AUTOMATION_COMPONENT_TEST_SCENARIO.CONTROLLER_PLUGIN_RECOVERY
	);
	_ResetAndRecoverIgnoreExceptionPolicy : AutomationComponentTestCase(
		name := "TestResetAndRecoverIgnoreExceptionPolicy",
		parent := THIS^,
		scenario := AUTOMATION_COMPONENT_TEST_SCENARIO.RESET_AND_RECOVER_IGNORE_EXCEPTION_POLICY
	);
	_AfterChildrenInitializingAndTimeoutPropagation : AutomationComponentTestCase(
		name := "TestAfterChildrenInitializingAndTimeoutPropagation",
		parent := THIS^,
		scenario := AUTOMATION_COMPONENT_TEST_SCENARIO.AFTER_CHILDREN_INITIALIZING_AND_TIMEOUT_PROPAGATION
	);
	_DisabledChildStopResetAndHmiCommandConsumption : AutomationComponentTestCase(
		name := "TestDisabledChildStopResetAndHmiCommandConsumption",
		parent := THIS^,
		scenario := AUTOMATION_COMPONENT_TEST_SCENARIO.DISABLED_CHILD_STOP_RESET_AND_HMI_COMMAND_CONSUMPTION
	);
END_VAR
VAR
	_Children : ARRAY [0.._ChildCount - 1] OF TOF_Testing.ITestElement :=
	[
		_LifecycleTransitions,
		_InitializationTimeout,
		_EnableDisable,
		_ChildErrorPolicyIgnore,
		_ChildErrorPolicySetErrorAndContinue,
		_ChildErrorPolicySetErrorAndStop,
		_EventBubbling,
		_EventBubblingStopPropagation,
		_EventBroadcasting,
		_InputOutputPhases,
		_OutputPhaseStop,
		_InputPhaseStop,
		_OutputPhaseContinuation,
		_PrimaryErrorBeforeLogging,
		_RunnerHappyPath,
		_RunnerNullComponentGuard,
		_ResetChildPolicies,
		_ResetFromStoppedHook,
		_ParentValidation,
		_DuplicateChild,
		_MismatchedChildParent,
		_InitializationFailureResult,
		_IndexedLookupContainment,
		_ControllerPluginRecovery,
		_ResetAndRecoverIgnoreExceptionPolicy,
		_AfterChildrenInitializingAndTimeoutPropagation,
		_DisabledChildStopResetAndHmiCommandConsumption
	];
END_VAR

(*!
<summary>Borrows the persistent case array. Callers must not modify it.</summary>
*)
{attribute 'monitoring' := 'call'}
PROPERTY Children : REFERENCE TO ARRAY [0.._ChildCount - 1] OF TOF_Testing.ITestElement
GET
Children REF= _Children;
END_GET
END_PROPERTY

(*!
<summary>Borrows the concrete class name. Callers must not modify it.</summary>
*)
{attribute 'monitoring' := 'call'}
PROPERTY ClassName : REFERENCE TO STRING
GET
ClassName REF= _ClassName;
END_GET
END_PROPERTY

(*!
<summary>Borrows the project namespace name. Callers must not modify it.</summary>
*)
{attribute 'monitoring' := 'call'}
PROPERTY NamespaceName : REFERENCE TO STRING
GET
NamespaceName REF= CurrentNamespace.Name;
END_GET
END_PROPERTY

(*!
<summary>Reports the complete instance size in bytes.</summary>
*)
{attribute 'monitoring' := 'call'}
PROPERTY SelfSize : ULINT
GET
SelfSize := XSIZEOF(THIS^);
END_GET
END_PROPERTY

END_FUNCTION_BLOCK

// ---- Tests/Automation/AutomationComponentTestCase.TcPOU
(*
SPDX-FileCopyrightText: © 2026 Oleksandr Tiutyk <trofimich@gmail.com>
SPDX-License-Identifier: MIT
License: https://opensource.org/license/mit
*)

(*!
<summary>Runs one automation component scenario in an isolated fixture.</summary>
<description>
Owns a freshly allocated fixture for the active run. AfterTest releases it after success or a reported
exception. A concrete pointer preserves FB_exit for the fixture and its nested resource owners.
Use one task. Do not copy the test case while it owns a fixture.
</description>
*)

{attribute 'no_assign'}
{attribute 'no_explicit_call' := 'do not call this function block directly'}
FUNCTION_BLOCK AutomationComponentTestCase EXTENDS TOF_Testing.SingleCycleTest
VAR_STAT
	{attribute 'hide'}
	_ClassName : STRING := __POUNAME();
END_VAR
VAR
	_Scenario : AUTOMATION_COMPONENT_TEST_SCENARIO;
	_Fixture : POINTER TO AutomationComponentTestFixture;
END_VAR

(*!
<summary>Selects the scenario without allocating its fixture.</summary>
<param name="name">Name reported for this case.</param>
<param name="parent">Group that owns this case.</param>
<param name="scenario">Scenario selected for the case.</param>
*)
METHOD FB_init : BOOL
VAR_INPUT
	bInitRetains: BOOL; // TRUE: the retain variables are initialized (reset warm / reset cold)
	bInCopyCode: BOOL; // TRUE: the instance will be copied to the copy code afterward (online change)
	name : WSTRING;
	parent : TOF_Testing.ITestElement;
	scenario : AUTOMATION_COMPONENT_TEST_SCENARIO;
END_VAR
IF NOT bInCopyCode THEN
	_Scenario := scenario;
END_IF

FB_init := TRUE;
END_METHOD

(*!
<summary>Allocates a fresh fixture and runs the selected scenario.</summary>
<description>Terminal allocation failure is raised at the task boundary after case handling.</description>
*)
METHOD PROTECTED ExecuteTest
VAR
	assertions : REFERENCE TO TOF_Testing.Assertions;
END_VAR
_Fixture := __NEW(AutomationComponentTestFixture);

IF _Fixture = 0 THEN
	TOF_Core.DynamicMemoryManager.RaiseAllocationFailure();

	RETURN;
END_IF

assertions REF= Assert;
_Fixture^.ExecuteScenario(scenario := _Scenario, assertions := assertions);
END_METHOD

(*!
<summary>Releases the fixture before the case outcome is published.</summary>
<description>The framework records an exception from teardown. Clear the stored alias before releasing.</description>
*)
METHOD PROTECTED AfterTest
VAR
	fixture : POINTER TO AutomationComponentTestFixture;
END_VAR
fixture := _Fixture;
_Fixture := 0;

IF fixture <> 0 THEN
	__DELETE(fixture);
END_IF
END_METHOD

(*!
<summary>Releases an active fixture if the case is unloaded before its teardown.</summary>
<description>The fixture and its nested FB_exit paths complete without exceptions.</description>
<param name="bInCopyCode">TwinCAT copy-code exit marker. The previous instance leaves copied storage alive.</param>
*)
METHOD FB_exit : BOOL
VAR_INPUT
	bInCopyCode : BOOL;
END_VAR
IF NOT bInCopyCode AND_THEN _Fixture <> 0 THEN
	__DELETE(_Fixture);
END_IF

FB_exit := TRUE;
END_METHOD

(*!
<summary>Borrows the concrete class name. Callers must not modify it.</summary>
*)
{attribute 'monitoring' := 'call'}
PROPERTY ClassName : REFERENCE TO STRING
GET
ClassName REF= _ClassName;
END_GET
END_PROPERTY

(*!
<summary>Borrows the project namespace name. Callers must not modify it.</summary>
*)
{attribute 'monitoring' := 'call'}
PROPERTY NamespaceName : REFERENCE TO STRING
GET
NamespaceName REF= CurrentNamespace.Name;
END_GET
END_PROPERTY

(*!
<summary>Reports the complete instance size in bytes.</summary>
*)
{attribute 'monitoring' := 'call'}
PROPERTY SelfSize : ULINT
GET
SelfSize := XSIZEOF(THIS^);
END_GET
END_PROPERTY

END_FUNCTION_BLOCK

// ---- Tests/Automation/AutomationComponentTestFixture.TcPOU
(*
SPDX-FileCopyrightText: © 2026 Oleksandr Tiutyk <trofimich@gmail.com>
SPDX-License-Identifier: MIT
License: https://opensource.org/license/mit
*)

(*!
<summary>Owns the state used by one automation component test scenario.</summary>
<description>
Each fixture starts with freshly constructed function blocks and stores no borrowed assertion context.
Owns synthetic parent and child components. The timed initialization case retains the fixture between scans.
The dedicated runner task publishes its own diagnostics. This fixture does not own those observations.
</description>
*)

{attribute 'enable_dynamic_creation'}
{attribute 'no_assign'}
{attribute 'no_explicit_call' := 'do not call this function block directly'}
FUNCTION_BLOCK AutomationComponentTestFixture
VAR_STAT
	{attribute 'hide'}
	_ClassName : STRING := __POUNAME();
END_VAR
VAR
	//! <summary>Persistent parent dependency for the initialization-timeout composite.</summary>
	_TimeoutRoot : MockAutomationController(name := "TimeoutRoot");
	//! <summary>Persistent composite borrowing the suite-owned root throughout the timeout scenario.</summary>
	_TimeoutComposite : MockCompositeAutomationComponent(name := "CompTimeout", parent := _TimeoutRoot);

	// Component fixtures live with the owning scenario instance.
	_ResetIgnoreBranch : MockCompositeAutomationComponent(name := "ResetIgnore", parent := _TimeoutRoot);
	_ResetContinueBranch : MockCompositeAutomationComponent(name := "ResetContinue", parent := _TimeoutRoot);
	_ResetStopBranch : MockCompositeAutomationComponent(name := "ResetStop", parent := _TimeoutRoot);

	_OrphanReadyLeaf : MockLeafAutomationComponent(name := "OrphanReadyLeaf", parent := 0);
	_OrphanPendingLeaf : MockLeafAutomationComponent(name := "OrphanPendingLeaf", parent := 0);
	_OrphanReadyBranch : MockCompositeAutomationComponent(name := "OrphanReadyBranch", parent := 0);
	_OrphanPendingBranch : MockCompositeAutomationComponent(name := "OrphanPendingBranch", parent := 0);
	_ValidPendingLeaf : MockLeafAutomationComponent(name := "ValidPendingLeaf", parent := _TimeoutRoot);
	_EmptyRoot : MockAutomationController(name := "EmptyRoot");

	_FirstNullBranch : MockCompositeAutomationComponent(name := "FirstNull", parent := _TimeoutRoot);
	_SecondNullBranch : MockCompositeAutomationComponent(name := "SecondNull", parent := _TimeoutRoot);
	_ThrowingChildBranch : MockCompositeAutomationComponent(name := "ThrowingChild", parent := _TimeoutRoot);
	_FailureOuterBranch : MockCompositeAutomationComponent(name := "OuterBranch", parent := _TimeoutRoot);
	_FailureInnerBranch : MockCompositeAutomationComponent(name := "InnerBranch", parent := _FailureOuterBranch);

	_LookupComposite : MockCompositeAutomationComponent(name := "LookupComposite", parent := _TimeoutRoot);
	_LookupController : MockPluginAutomationController(name := "LookupController");

	_HmiPlugin : MockHmiControllerPlugin;
	_HmiPlugins : ARRAY [0..0] OF TOF_Automation.IAutomationControllerPlugin := [_HmiPlugin];
	_HmiController : MockPluginAutomationController(name := "HmiController");
	_InvalidHmiController : MockPluginAutomationController(name := "InvalidHmiController");

	_OutputStopBranch : MockCompositeAutomationComponent(name := "OutputBranch", parent := _TimeoutRoot);
	_OutputStopController : MockPluginAutomationController(name := "OutputController");

